Yaskawa INFORM job: vendrediTRJ3.JBI

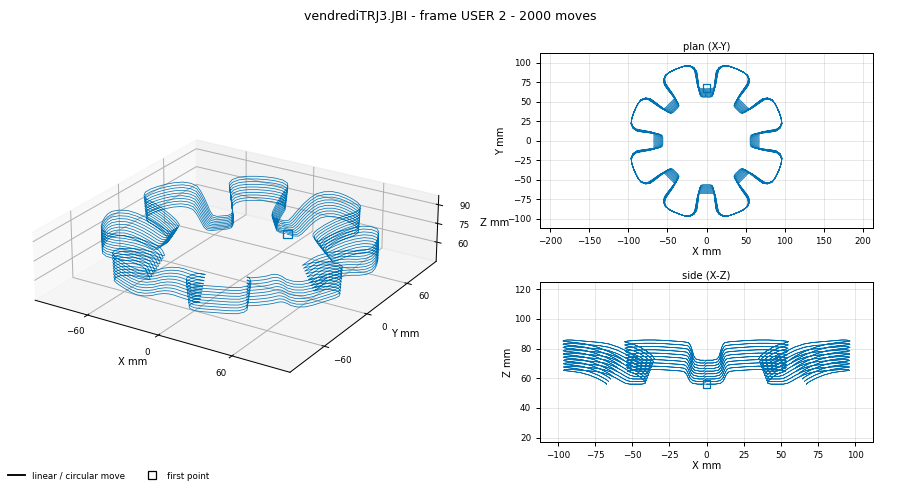
[picture p0: tool path of vendrediTRJ3.JBI in frame USER 2, 2000 of 2000 moves have a stored position in this frame; points joined in program order, loops and branches not executed]
/JOB
//NAME temp/vendrediTRJ3
///FOLDERNAME DEMO
//POS
///NPOS 2000,0,2000,0,0,0
///USER 2
///TOOL 7
///POSTYPE USER
///RECTAN
///RCONF 1,0,0,0,0,0,0,0,0,0,0,0,0,0,0,0,0,0,0,0,0,0,0,0
C00000=0.000,67.469,56.061,180.0000,38.4594,-10890.0000
C00001=2.820,67.413,56.044,-179.6998,38.4717,-10892.3954
C00002=5.989,67.263,56.069,174.6494,37.7561,-10895.0881
C00003=9.441,67.734,56.637,160.4399,22.8847,-10897.9350
C00004=11.191,69.937,58.076,177.3917,0.4478,-10899.0911
C00005=12.227,73.809,60.085,-176.5319,-0.2393,-10899.4060
C00006=13.183,79.025,62.181,-173.7887,-0.2511,-10899.4709
C00007=14.211,84.918,63.804,-172.0889,-0.3684,-10899.5004
C00008=15.500,90.396,64.610,-172.2474,-1.9783,-10899.7298
C00009=18.832,94.373,65.037,-176.4691,-3.4890,-10901.2851
C00010=23.832,96.213,65.385,-179.1427,-2.3150,-10903.9122
C00011=29.513,95.497,65.736,-179.9981,-0.1613,-10907.1736
C00012=35.347,93.539,65.969,-179.9993,-0.0181,-10910.7008
C00013=41.148,91.136,65.969,-179.9981,-0.0180,-10914.2992
C00014=46.658,88.395,65.736,179.9983,-0.1564,-10917.8267
C00015=51.181,84.885,65.385,179.1465,-2.3148,-10921.0877
C00016=53.416,80.048,65.037,176.4667,-3.4903,-10923.7152
C00017=52.959,74.880,64.610,172.2446,-1.9818,-10925.2699
C00018=49.997,70.095,63.804,172.0881,-0.3719,-10925.4993
C00019=46.557,65.200,62.181,173.7887,-0.2530,-10925.5293
C00020=43.545,60.837,60.085,176.5334,-0.2396,-10925.5938
C00021=41.540,57.367,58.076,-177.3875,0.4483,-10925.9087
C00022=41.220,54.571,56.637,-160.4399,22.8842,-10927.0654
C00023=43.327,51.796,56.069,-174.6518,37.7544,-10929.9123
C00024=45.674,49.662,56.044,179.7031,38.4687,-10932.6047
C00025=47.708,47.708,56.061,-180.0000,38.4581,-10935.0000
C00026=49.662,45.674,56.044,-179.7031,38.4687,-10937.3953
C00027=51.797,43.327,56.069,174.6514,37.7543,-10940.0883
C00028=54.571,41.220,56.637,160.4399,22.8842,-10942.9346
C00029=57.367,41.540,58.076,177.3875,0.4483,-10944.0913
C00030=60.837,43.545,60.085,-176.5334,-0.2396,-10944.4062
C00031=65.200,46.557,62.181,-173.7887,-0.2530,-10944.4707
C00032=70.095,49.997,63.804,-172.0881,-0.3719,-10944.5007
C00033=74.880,52.959,64.610,-172.2446,-1.9818,-10944.7301
C00034=80.048,53.416,65.037,-176.4667,-3.4903,-10946.2848
C00035=84.885,51.181,65.385,-179.1465,-2.3148,-10948.9123
C00036=88.395,46.658,65.736,-179.9983,-0.1564,-10952.1733
C00037=91.136,41.148,65.969,179.9981,-0.0180,-10955.7008
C00038=93.539,35.347,65.969,179.9993,-0.0181,-10959.2992
C00039=95.497,29.513,65.736,179.9981,-0.1613,-10962.8264
C00040=96.213,23.832,65.385,179.1427,-2.3150,-10966.0878
C00041=94.373,18.832,65.037,176.4691,-3.4890,-10968.7149
C00042=90.396,15.500,64.610,172.2474,-1.9783,-10970.2702
C00043=84.918,14.211,63.804,172.0889,-0.3684,-10970.4996
C00044=79.025,13.183,62.181,173.7887,-0.2511,-10970.5291
C00045=73.809,12.227,60.085,176.5319,-0.2393,-10970.5940
C00046=69.937,11.191,58.076,-177.3917,0.4478,-10970.9089
C00047=67.734,9.441,56.637,-160.4399,22.8847,-10972.0650
C00048=67.263,5.989,56.069,-174.6494,37.7561,-10974.9119
C00049=67.413,2.820,56.044,179.6998,38.4717,-10977.6046
C00050=67.469,0.000,56.061,-180.0000,38.4594,-10980.0000
C00051=67.413,-2.820,56.044,-179.6998,38.4717,-10982.3954
C00052=67.263,-5.989,56.069,174.6494,37.7561,-10985.0881
C00053=67.734,-9.441,56.637,160.4399,22.8847,-10987.9350
C00054=69.937,-11.191,58.076,177.3917,0.4478,-10989.0911
C00055=73.809,-12.227,60.085,-176.5319,-0.2393,-10989.4060
C00056=79.025,-13.183,62.181,-173.7887,-0.2511,-10989.4709
C00057=84.918,-14.211,63.804,-172.0889,-0.3684,-10989.5004
C00058=90.396,-15.500,64.610,-172.2474,-1.9783,-10989.7298
C00059=94.373,-18.832,65.037,-176.4691,-3.4890,-10991.2851
C00060=96.213,-23.832,65.385,-179.1427,-2.3150,-10993.9122
C00061=95.497,-29.513,65.736,-179.9981,-0.1613,-10997.1736
C00062=93.539,-35.347,65.969,-179.9993,-0.0181,-11000.7008
C00063=91.136,-41.148,65.969,-179.9981,-0.0180,-11004.2992
C00064=88.395,-46.658,65.736,179.9983,-0.1564,-11007.8267
C00065=84.885,-51.181,65.385,179.1465,-2.3148,-11011.0877
C00066=80.048,-53.416,65.037,176.4667,-3.4903,-11013.7152
C00067=74.880,-52.959,64.610,172.2446,-1.9818,-11015.2699
C00068=70.095,-49.997,63.804,172.0881,-0.3719,-11015.4993
C00069=65.200,-46.557,62.181,173.7887,-0.2530,-11015.5293
C00070=60.837,-43.545,60.085,176.5334,-0.2396,-11015.5938
C00071=57.367,-41.540,58.076,-177.3875,0.4483,-11015.9087
C00072=54.571,-41.220,56.637,-160.4399,22.8842,-11017.0654
C00073=51.796,-43.327,56.069,-174.6518,37.7544,-11019.9123
C00074=49.662,-45.674,56.044,179.7031,38.4687,-11022.6047
C00075=47.708,-47.708,56.061,-180.0000,38.4581,-11025.0000
C00076=45.674,-49.662,56.044,-179.7031,38.4687,-11027.3953
C00077=43.327,-51.797,56.069,174.6514,37.7543,-11030.0883
C00078=41.220,-54.571,56.637,160.4399,22.8842,-11032.9346
C00079=41.540,-57.367,58.076,177.3875,0.4483,-11034.0913
C00080=43.545,-60.837,60.085,-176.5334,-0.2396,-11034.4062
C00081=46.557,-65.200,62.181,-173.7887,-0.2530,-11034.4707
C00082=49.997,-70.095,63.804,-172.0881,-0.3719,-11034.5007
C00083=52.959,-74.880,64.610,-172.2446,-1.9818,-11034.7301
C00084=53.416,-80.048,65.037,-176.4667,-3.4903,-11036.2848
C00085=51.181,-84.885,65.385,-179.1465,-2.3148,-11038.9123
C00086=46.658,-88.395,65.736,-179.9983,-0.1564,-11042.1733
C00087=41.148,-91.136,65.969,179.9981,-0.0180,-11045.7008
C00088=35.347,-93.539,65.969,179.9993,-0.0181,-11049.2992
C00089=29.513,-95.497,65.736,179.9981,-0.1613,-11052.8264
C00090=23.832,-96.213,65.385,179.1427,-2.3150,-11056.0878
C00091=18.832,-94.373,65.037,176.4691,-3.4890,-11058.7149
C00092=15.500,-90.396,64.610,172.2474,-1.9783,-11060.2702
C00093=14.211,-84.918,63.804,172.0889,-0.3684,-11060.4996
C00094=13.183,-79.025,62.181,173.7887,-0.2511,-11060.5291
C00095=12.227,-73.809,60.085,176.5319,-0.2393,-11060.5940
C00096=11.191,-69.937,58.076,-177.3917,0.4478,-11060.9089
C00097=9.441,-67.734,56.637,-160.4399,22.8847,-11062.0650
C00098=5.989,-67.263,56.069,-174.6494,37.7561,-11064.9119
C00099=2.820,-67.413,56.044,179.6998,38.4717,-11067.6046
C00100=0.000,-67.469,56.061,-180.0000,38.4594,-11070.0000
C00101=-2.820,-67.413,56.044,-179.6998,38.4717,-11072.3954
C00102=-5.989,-67.263,56.069,174.6494,37.7561,-11075.0881
C00103=-9.441,-67.734,56.637,160.4399,22.8847,-11077.9350
C00104=-11.191,-69.937,58.076,177.3917,0.4478,-11079.0911
C00105=-12.227,-73.809,60.085,-176.5319,-0.2393,-11079.4060
C00106=-13.183,-79.025,62.181,-173.7887,-0.2511,-11079.4709
C00107=-14.211,-84.918,63.804,-172.0889,-0.3684,-11079.5004
C00108=-15.500,-90.396,64.610,-172.2474,-1.9783,-11079.7298
C00109=-18.832,-94.373,65.037,-176.4691,-3.4890,-11081.2851
C00110=-23.832,-96.213,65.385,-179.1427,-2.3150,-11083.9122
C00111=-29.513,-95.497,65.736,-179.9981,-0.1613,-11087.1736
C00112=-35.347,-93.539,65.969,-179.9993,-0.0181,-11090.7008
C00113=-41.148,-91.136,65.969,-179.9981,-0.0180,-11094.2992
C00114=-46.658,-88.395,65.736,179.9983,-0.1564,-11097.8267
C00115=-51.181,-84.885,65.385,179.1465,-2.3148,-11101.0877
C00116=-53.416,-80.048,65.037,176.4667,-3.4903,-11103.7152
C00117=-52.959,-74.880,64.610,172.2446,-1.9818,-11105.2699
C00118=-49.997,-70.095,63.804,172.0881,-0.3719,-11105.4993
C00119=-46.557,-65.200,62.181,173.7887,-0.2530,-11105.5293
C00120=-43.545,-60.837,60.085,176.5334,-0.2396,-11105.5938
C00121=-41.540,-57.367,58.076,-177.3875,0.4483,-11105.9087
C00122=-41.220,-54.571,56.637,-160.4399,22.8842,-11107.0654
C00123=-43.327,-51.796,56.069,-174.6518,37.7544,-11109.9123
C00124=-45.674,-49.662,56.044,179.7031,38.4687,-11112.6047
C00125=-47.708,-47.708,56.061,-180.0000,38.4581,-11115.0000
C00126=-49.662,-45.674,56.044,-179.7031,38.4687,-11117.3953
C00127=-51.797,-43.327,56.069,174.6514,37.7543,-11120.0883
C00128=-54.571,-41.220,56.637,160.4399,22.8842,-11122.9346
C00129=-57.367,-41.540,58.076,177.3875,0.4483,-11124.0913
C00130=-60.837,-43.545,60.085,-176.5334,-0.2396,-11124.4062
C00131=-65.200,-46.557,62.181,-173.7887,-0.2530,-11124.4707
C00132=-70.095,-49.997,63.804,-172.0881,-0.3719,-11124.5007
C00133=-74.880,-52.959,64.610,-172.2446,-1.9818,-11124.7301
C00134=-80.048,-53.416,65.037,-176.4667,-3.4903,-11126.2848
C00135=-84.885,-51.181,65.385,-179.1465,-2.3148,-11128.9123
C00136=-88.395,-46.658,65.736,-179.9983,-0.1564,-11132.1733
C00137=-91.136,-41.148,65.969,179.9981,-0.0180,-11135.7008
C00138=-93.539,-35.347,65.969,179.9993,-0.0181,-11139.2992
C00139=-95.497,-29.513,65.736,179.9981,-0.1613,-11142.8264
C00140=-96.213,-23.832,65.385,179.1427,-2.3150,-11146.0878
C00141=-94.373,-18.832,65.037,176.4691,-3.4890,-11148.7149
C00142=-90.396,-15.500,64.610,172.2474,-1.9783,-11150.2702
C00143=-84.918,-14.211,63.804,172.0889,-0.3684,-11150.4996
C00144=-79.025,-13.183,62.181,173.7887,-0.2511,-11150.5291
C00145=-73.809,-12.227,60.085,176.5319,-0.2393,-11150.5940
C00146=-69.937,-11.191,58.076,-177.3917,0.4478,-11150.9089
C00147=-67.734,-9.441,56.637,-160.4399,22.8847,-11152.0650
C00148=-67.263,-5.989,56.069,-174.6494,37.7561,-11154.9119
C00149=-67.413,-2.820,56.044,179.6998,38.4717,-11157.6046
C00150=-67.469,0.000,56.061,-180.0000,38.4594,-11160.0000
C00151=-67.413,2.820,56.044,-179.6998,38.4717,-11162.3954
C00152=-67.263,5.989,56.069,174.6494,37.7561,-11165.0881
C00153=-67.734,9.441,56.637,160.4399,22.8847,-11167.9350
C00154=-69.937,11.191,58.076,177.3917,0.4478,-11169.0911
C00155=-73.809,12.227,60.085,-176.5319,-0.2393,-11169.4060
C00156=-79.025,13.183,62.181,-173.7887,-0.2511,-11169.4709
C00157=-84.918,14.211,63.804,-172.0889,-0.3684,-11169.5004
C00158=-90.396,15.500,64.610,-172.2474,-1.9783,-11169.7298
C00159=-94.373,18.832,65.037,-176.4691,-3.4890,-11171.2851
C00160=-96.213,23.832,65.385,-179.1427,-2.3150,-11173.9122
C00161=-95.497,29.513,65.736,-179.9981,-0.1613,-11177.1736
C00162=-93.539,35.347,65.969,-179.9993,-0.0181,-11180.7008
C00163=-91.136,41.148,65.969,-179.9981,-0.0180,-11184.2992
C00164=-88.395,46.658,65.736,179.9983,-0.1564,-11187.8267
C00165=-84.885,51.181,65.385,179.1465,-2.3148,-11191.0877
C00166=-80.048,53.416,65.037,176.4667,-3.4903,-11193.7152
C00167=-74.880,52.959,64.610,172.2446,-1.9818,-11195.2699
C00168=-70.095,49.997,63.804,172.0881,-0.3719,-11195.4993
C00169=-65.200,46.557,62.181,173.7887,-0.2530,-11195.5293
C00170=-60.837,43.545,60.085,176.5334,-0.2396,-11195.5938
C00171=-57.367,41.540,58.076,-177.3875,0.4483,-11195.9087
C00172=-54.571,41.220,56.637,-160.4399,22.8842,-11197.0654
C00173=-51.796,43.327,56.069,-174.6518,37.7544,-11199.9123
C00174=-49.662,45.674,56.044,179.7031,38.4687,-11202.6047
C00175=-47.708,47.708,56.061,-180.0000,38.4581,-11205.0000
C00176=-45.674,49.662,56.044,-179.7031,38.4687,-11207.3953
C00177=-43.327,51.797,56.069,174.6514,37.7543,-11210.0883
C00178=-41.220,54.571,56.637,160.4399,22.8842,-11212.9346
C00179=-41.540,57.367,58.076,177.3875,0.4483,-11214.0913
C00180=-43.545,60.837,60.085,-176.5334,-0.2396,-11214.4062
C00181=-46.557,65.200,62.181,-173.7887,-0.2530,-11214.4707
C00182=-49.997,70.095,63.804,-172.0881,-0.3719,-11214.5007
C00183=-52.959,74.880,64.610,-172.2446,-1.9818,-11214.7301
C00184=-53.416,80.048,65.037,-176.4667,-3.4903,-11216.2848
C00185=-51.181,84.885,65.385,-179.1465,-2.3148,-11218.9123
C00186=-46.658,88.395,65.736,-179.9983,-0.1564,-11222.1733
C00187=-41.148,91.136,65.969,179.9981,-0.0180,-11225.7008
C00188=-35.347,93.539,65.969,179.9993,-0.0181,-11229.2992
C00189=-29.513,95.497,65.736,179.9981,-0.1613,-11232.8264
C00190=-23.832,96.213,65.385,179.1427,-2.3150,-11236.0878
C00191=-18.832,94.373,65.037,176.4691,-3.4890,-11238.7149
C00192=-15.500,90.396,64.610,172.2474,-1.9783,-11240.2702
C00193=-14.211,84.918,63.804,172.0889,-0.3684,-11240.4996
C00194=-13.183,79.025,62.181,173.7887,-0.2511,-11240.5291
C00195=-12.227,73.809,60.085,176.5319,-0.2393,-11240.5940
C00196=-11.191,69.937,58.076,-177.3917,0.4478,-11240.9089
C00197=-9.441,67.734,56.637,-160.4399,22.8847,-11242.0650
C00198=-5.989,67.263,56.069,-174.6494,37.7561,-11244.9119
C00199=-2.820,67.413,56.044,179.6998,38.4717,-11247.6046
C00200=0.000,66.107,57.788,180.0000,38.0594,-11250.0000
C00201=2.695,66.055,57.771,-179.6967,38.0667,-11252.3363
C00202=5.779,65.917,57.797,174.4231,37.2903,-11255.0104
C00203=9.185,66.436,58.394,160.6412,21.4973,-11257.8714
C00204=10.880,68.762,59.909,178.2705,0.2602,-11258.9912
C00205=11.874,72.826,62.021,-176.2283,-0.2219,-11259.2604
C00206=12.805,78.288,64.219,-173.7529,-0.2122,-11259.2892
C00207=13.814,84.445,65.915,-172.1933,-0.3031,-11259.2905
C00208=15.073,90.163,66.756,-172.3373,-1.8422,-11259.4907
C00209=18.432,94.325,67.200,-176.4590,-3.4166,-11261.0568
C00210=23.517,96.271,67.561,-179.1417,-2.2803,-11263.7273
C00211=29.315,95.562,67.927,179.9999,-0.1559,-11267.0541
C00212=35.280,93.564,68.167,-179.9993,-0.0181,-11270.6599
C00213=41.213,91.107,68.167,-179.9981,-0.0180,-11274.3400
C00214=46.844,88.301,67.927,179.9986,-0.1564,-11277.9461
C00215=51.445,84.703,67.561,179.1429,-2.2773,-11281.2727
C00216=53.664,79.731,67.200,176.4564,-3.4170,-11283.9430
C00217=53.097,74.413,66.756,172.3397,-1.8459,-11285.5096
C00218=49.944,69.479,65.915,172.1917,-0.3060,-11285.7099
C00219=46.303,64.413,64.219,173.7509,-0.2085,-11285.7103
C00220=43.100,59.892,62.021,176.2254,-0.2229,-11285.7399
C00221=40.929,56.315,59.909,-178.2687,0.2595,-11286.0092
C00222=40.483,53.472,58.394,-160.6426,21.4997,-11287.1289
C00223=42.524,50.697,57.797,-174.4236,37.2887,-11289.9895
C00224=44.802,48.614,57.771,179.6988,38.0662,-11292.6632
C00225=46.745,46.745,57.788,180.0000,38.0574,-11295.0000
C00226=48.613,44.802,57.771,-179.6984,38.0662,-11297.3362
C00227=50.697,42.524,57.797,174.4190,37.2852,-11300.0105
C00228=53.472,40.483,58.395,160.6426,21.4997,-11302.8711
C00229=56.315,40.929,59.909,178.2687,0.2595,-11303.9908
C00230=59.892,43.100,62.021,-176.2254,-0.2229,-11304.2601
C00231=64.413,46.303,64.219,-173.7509,-0.2085,-11304.2897
C00232=69.479,49.944,65.915,-172.1917,-0.3060,-11304.2901
C00233=74.413,53.097,66.756,-172.3397,-1.8459,-11304.4904
C00234=79.731,53.664,67.200,-176.4564,-3.4170,-11306.0570
C00235=84.703,51.445,67.561,-179.1429,-2.2773,-11308.7273
C00236=88.301,46.844,67.927,-179.9986,-0.1564,-11312.0539
C00237=91.107,41.213,68.167,179.9981,-0.0180,-11315.6600
C00238=93.564,35.280,68.167,179.9993,-0.0181,-11319.3401
C00239=95.562,29.315,67.927,-179.9999,-0.1559,-11322.9459
C00240=96.271,23.517,67.561,179.1417,-2.2803,-11326.2727
C00241=94.325,18.432,67.200,176.4590,-3.4166,-11328.9432
C00242=90.163,15.073,66.756,172.3373,-1.8422,-11330.5093
C00243=84.445,13.814,65.915,172.1933,-0.3031,-11330.7095
C00244=78.288,12.805,64.219,173.7529,-0.2122,-11330.7108
C00245=72.826,11.874,62.021,176.2283,-0.2219,-11330.7396
C00246=68.762,10.880,59.909,-178.2705,0.2602,-11331.0088
C00247=66.436,9.185,58.394,-160.6412,21.4973,-11332.1286
C00248=65.917,5.779,57.797,-174.4231,37.2903,-11334.9896
C00249=66.055,2.695,57.771,179.6967,38.0667,-11337.6637
C00250=66.107,0.000,57.788,180.0000,38.0594,-11340.0000
C00251=66.055,-2.695,57.771,-179.6967,38.0667,-11342.3363
C00252=65.917,-5.780,57.797,174.4154,37.2898,-11345.0112
C00253=66.436,-9.185,58.395,160.6412,21.4973,-11347.8714
C00254=68.762,-10.880,59.909,178.2705,0.2602,-11348.9912
C00255=72.826,-11.874,62.021,-176.2283,-0.2219,-11349.2604
C00256=78.288,-12.805,64.219,-173.7529,-0.2122,-11349.2892
C00257=84.445,-13.814,65.915,-172.1933,-0.3031,-11349.2905
C00258=90.163,-15.073,66.756,-172.3373,-1.8422,-11349.4907
C00259=94.325,-18.432,67.200,-176.4590,-3.4166,-11351.0568
C00260=96.271,-23.517,67.561,-179.1417,-2.2803,-11353.7273
C00261=95.562,-29.315,67.927,179.9999,-0.1559,-11357.0541
C00262=93.564,-35.280,68.167,-179.9993,-0.0181,-11360.6599
C00263=91.107,-41.213,68.167,-179.9981,-0.0180,-11364.3400
C00264=88.301,-46.844,67.927,179.9986,-0.1564,-11367.9461
C00265=84.703,-51.445,67.561,179.1429,-2.2773,-11371.2727
C00266=79.731,-53.664,67.200,176.4564,-3.4170,-11373.9430
C00267=74.413,-53.097,66.756,172.3397,-1.8459,-11375.5096
C00268=69.479,-49.944,65.915,172.1917,-0.3060,-11375.7099
C00269=64.413,-46.303,64.219,173.7509,-0.2085,-11375.7103
C00270=59.892,-43.100,62.021,176.2254,-0.2229,-11375.7399
C00271=56.315,-40.929,59.909,-178.2687,0.2595,-11376.0092
C00272=53.472,-40.483,58.394,-160.6426,21.4997,-11377.1289
C00273=50.697,-42.524,57.797,-174.4236,37.2887,-11379.9895
C00274=48.614,-44.802,57.771,179.6988,38.0662,-11382.6632
C00275=46.745,-46.745,57.788,180.0000,38.0574,-11385.0000
C00276=44.802,-48.613,57.771,-179.6984,38.0662,-11387.3362
C00277=42.524,-50.697,57.797,174.4190,37.2852,-11390.0105
C00278=40.483,-53.472,58.395,160.6426,21.4997,-11392.8711
C00279=40.929,-56.315,59.909,178.2687,0.2595,-11393.9908
C00280=43.100,-59.892,62.021,-176.2254,-0.2229,-11394.2601
C00281=46.303,-64.413,64.219,-173.7509,-0.2085,-11394.2897
C00282=49.944,-69.479,65.915,-172.1917,-0.3060,-11394.2901
C00283=53.097,-74.413,66.756,-172.3397,-1.8459,-11394.4904
C00284=53.664,-79.731,67.200,-176.4564,-3.4170,-11396.0570
C00285=51.445,-84.703,67.561,-179.1429,-2.2773,-11398.7273
C00286=46.844,-88.301,67.927,-179.9986,-0.1564,-11402.0539
C00287=41.213,-91.107,68.167,179.9981,-0.0180,-11405.6600
C00288=35.280,-93.564,68.167,179.9993,-0.0181,-11409.3401
C00289=29.315,-95.562,67.927,-179.9999,-0.1559,-11412.9459
C00290=23.517,-96.271,67.561,179.1417,-2.2803,-11416.2727
C00291=18.432,-94.325,67.200,176.4590,-3.4166,-11418.9432
C00292=15.073,-90.163,66.756,172.3373,-1.8422,-11420.5093
C00293=13.814,-84.445,65.915,172.1933,-0.3031,-11420.7095
C00294=12.805,-78.288,64.219,173.7529,-0.2122,-11420.7108
C00295=11.874,-72.826,62.021,176.2283,-0.2219,-11420.7396
C00296=10.880,-68.762,59.909,-178.2705,0.2602,-11421.0088
C00297=9.185,-66.436,58.394,-160.6412,21.4973,-11422.1286
C00298=5.779,-65.917,57.797,-174.4231,37.2903,-11424.9896
C00299=2.695,-66.055,57.771,179.6967,38.0667,-11427.6637
C00300=0.000,-66.107,57.788,-180.0000,38.0594,-11430.0000
C00301=-2.695,-66.055,57.771,-179.6967,38.0667,-11432.3363
C00302=-5.780,-65.917,57.797,174.4154,37.2898,-11435.0112
C00303=-9.185,-66.436,58.395,160.6412,21.4973,-11437.8714
C00304=-10.880,-68.762,59.909,178.2705,0.2602,-11438.9912
C00305=-11.874,-72.826,62.021,-176.2283,-0.2219,-11439.2604
C00306=-12.805,-78.288,64.219,-173.7529,-0.2122,-11439.2892
C00307=-13.814,-84.445,65.915,-172.1933,-0.3031,-11439.2905
C00308=-15.073,-90.163,66.756,-172.3373,-1.8422,-11439.4907
C00309=-18.432,-94.325,67.200,-176.4590,-3.4166,-11441.0568
C00310=-23.517,-96.271,67.561,-179.1417,-2.2803,-11443.7273
C00311=-29.315,-95.562,67.927,179.9999,-0.1559,-11447.0541
C00312=-35.280,-93.564,68.167,-179.9993,-0.0181,-11450.6599
C00313=-41.213,-91.107,68.167,-179.9981,-0.0180,-11454.3400
C00314=-46.844,-88.301,67.927,179.9986,-0.1564,-11457.9461
C00315=-51.445,-84.703,67.561,179.1429,-2.2773,-11461.2727
C00316=-53.664,-79.731,67.200,176.4564,-3.4170,-11463.9430
C00317=-53.097,-74.413,66.756,172.3397,-1.8459,-11465.5096
C00318=-49.944,-69.479,65.915,172.1917,-0.3060,-11465.7099
C00319=-46.303,-64.413,64.219,173.7509,-0.2085,-11465.7103
C00320=-43.100,-59.892,62.021,176.2254,-0.2229,-11465.7399
C00321=-40.929,-56.315,59.909,-178.2687,0.2595,-11466.0092
C00322=-40.483,-53.472,58.394,-160.6426,21.4997,-11467.1289
C00323=-42.524,-50.697,57.797,-174.4236,37.2887,-11469.9895
C00324=-44.802,-48.614,57.771,179.6988,38.0662,-11472.6632
C00325=-46.745,-46.745,57.788,-180.0000,38.0574,-11475.0000
C00326=-48.613,-44.802,57.771,-179.6984,38.0662,-11477.3362
C00327=-50.697,-42.524,57.797,174.4190,37.2852,-11480.0105
C00328=-53.472,-40.483,58.395,160.6426,21.4997,-11482.8711
C00329=-56.315,-40.929,59.909,178.2687,0.2595,-11483.9908
C00330=-59.892,-43.100,62.021,-176.2254,-0.2229,-11484.2601
C00331=-64.413,-46.303,64.219,-173.7509,-0.2085,-11484.2897
C00332=-69.479,-49.944,65.915,-172.1917,-0.3060,-11484.2901
C00333=-74.413,-53.097,66.756,-172.3397,-1.8459,-11484.4904
C00334=-79.731,-53.664,67.200,-176.4564,-3.4170,-11486.0570
C00335=-84.703,-51.445,67.561,-179.1429,-2.2773,-11488.7273
C00336=-88.301,-46.844,67.927,-179.9986,-0.1564,-11492.0539
C00337=-91.107,-41.213,68.167,179.9981,-0.0180,-11495.6600
C00338=-93.564,-35.280,68.167,179.9993,-0.0181,-11499.3401
C00339=-95.562,-29.315,67.927,-179.9999,-0.1559,-11502.9459
C00340=-96.271,-23.517,67.561,179.1417,-2.2803,-11506.2727
C00341=-94.325,-18.432,67.200,176.4590,-3.4166,-11508.9432
C00342=-90.163,-15.073,66.756,172.3373,-1.8422,-11510.5093
C00343=-84.445,-13.814,65.915,172.1933,-0.3031,-11510.7095
C00344=-78.288,-12.805,64.219,173.7529,-0.2122,-11510.7108
C00345=-72.826,-11.874,62.021,176.2283,-0.2219,-11510.7396
C00346=-68.762,-10.880,59.909,-178.2705,0.2602,-11511.0088
C00347=-66.436,-9.185,58.394,-160.6412,21.4973,-11512.1286
C00348=-65.917,-5.779,57.797,-174.4231,37.2903,-11514.9896
C00349=-66.055,-2.695,57.771,179.6967,38.0667,-11517.6637
C00350=-66.107,0.000,57.788,-180.0000,38.0594,-11520.0000
C00351=-66.055,2.695,57.771,-179.6967,38.0667,-11522.3363
C00352=-65.917,5.780,57.797,174.4154,37.2898,-11525.0112
C00353=-66.436,9.185,58.395,160.6412,21.4973,-11527.8714
C00354=-68.762,10.880,59.909,178.2705,0.2602,-11528.9912
C00355=-72.826,11.874,62.021,-176.2283,-0.2219,-11529.2604
C00356=-78.288,12.805,64.219,-173.7529,-0.2122,-11529.2892
C00357=-84.445,13.814,65.915,-172.1933,-0.3031,-11529.2905
C00358=-90.163,15.073,66.756,-172.3373,-1.8422,-11529.4907
C00359=-94.325,18.432,67.200,-176.4590,-3.4166,-11531.0568
C00360=-96.271,23.517,67.561,-179.1417,-2.2803,-11533.7273
C00361=-95.562,29.315,67.927,179.9999,-0.1559,-11537.0541
C00362=-93.564,35.280,68.167,-179.9993,-0.0181,-11540.6599
C00363=-91.107,41.213,68.167,-179.9981,-0.0180,-11544.3400
C00364=-88.301,46.844,67.927,179.9986,-0.1564,-11547.9461
C00365=-84.703,51.445,67.561,179.1429,-2.2773,-11551.2727
C00366=-79.731,53.664,67.200,176.4564,-3.4170,-11553.9430
C00367=-74.413,53.097,66.756,172.3397,-1.8459,-11555.5096
C00368=-69.479,49.944,65.915,172.1917,-0.3060,-11555.7099
C00369=-64.413,46.303,64.219,173.7509,-0.2085,-11555.7103
C00370=-59.892,43.100,62.021,176.2254,-0.2229,-11555.7399
C00371=-56.315,40.929,59.909,-178.2687,0.2595,-11556.0092
C00372=-53.472,40.483,58.394,-160.6426,21.4997,-11557.1289
C00373=-50.697,42.524,57.797,-174.4236,37.2887,-11559.9895
C00374=-48.614,44.802,57.771,179.6988,38.0662,-11562.6632
C00375=-46.745,46.745,57.788,-180.0000,38.0574,-11565.0000
C00376=-44.802,48.613,57.771,-179.6984,38.0662,-11567.3362
C00377=-42.524,50.697,57.797,174.4190,37.2852,-11570.0105
C00378=-40.483,53.472,58.395,160.6426,21.4997,-11572.8711
C00379=-40.929,56.315,59.909,178.2687,0.2595,-11573.9908
C00380=-43.100,59.892,62.021,-176.2254,-0.2229,-11574.2601
C00381=-46.303,64.413,64.219,-173.7509,-0.2085,-11574.2897
C00382=-49.944,69.479,65.915,-172.1917,-0.3060,-11574.2901
C00383=-53.097,74.413,66.756,-172.3397,-1.8459,-11574.4904
C00384=-53.664,79.731,67.200,-176.4564,-3.4170,-11576.0570
C00385=-51.445,84.703,67.561,-179.1429,-2.2773,-11578.7273
C00386=-46.844,88.301,67.927,-179.9986,-0.1564,-11582.0539
C00387=-41.213,91.107,68.167,179.9981,-0.0180,-11585.6600
C00388=-35.280,93.564,68.167,179.9993,-0.0181,-11589.3401
C00389=-29.315,95.562,67.927,-179.9999,-0.1559,-11592.9459
C00390=-23.517,96.271,67.561,179.1417,-2.2803,-11596.2727
C00391=-18.432,94.325,67.200,176.4590,-3.4166,-11598.9432
C00392=-15.073,90.163,66.756,172.3373,-1.8422,-11600.5093
C00393=-13.814,84.445,65.915,172.1933,-0.3031,-11600.7095
C00394=-12.805,78.288,64.219,173.7529,-0.2122,-11600.7108
C00395=-11.874,72.826,62.021,176.2283,-0.2219,-11600.7396
C00396=-10.880,68.762,59.909,-178.2705,0.2602,-11601.0088
C00397=-9.185,66.436,58.395,-160.6412,21.4973,-11602.1286
C00398=-5.780,65.917,57.797,-174.4154,37.2898,-11604.9888
C00399=-2.695,66.055,57.771,179.6967,38.0667,-11607.6637
C00400=0.000,64.758,59.526,-180.0000,37.5735,-11610.0000
C00401=2.572,64.710,59.508,-179.6979,37.5837,-11612.2761
C00402=5.572,64.584,59.535,174.2146,36.7296,-11614.9310
C00403=8.932,65.152,60.163,160.9703,20.0908,-11617.8063
C00404=10.572,67.603,61.754,179.0583,0.1253,-11618.8881
C00405=11.527,71.864,63.969,-175.9897,-0.1992,-11619.1126
C00406=12.439,77.571,66.266,-173.7747,-0.1711,-11619.1102
C00407=13.430,83.988,68.033,-172.3612,-0.2407,-11619.0849
C00408=14.662,89.940,68.906,-172.5060,-1.7115,-11619.2589
C00409=18.048,94.279,69.366,-176.4898,-3.3102,-11620.8371
C00410=23.215,96.325,69.740,-179.1510,-2.2246,-11623.5503
C00411=29.126,95.625,70.117,179.9996,-0.1559,-11626.9400
C00412=35.216,93.589,70.366,-179.9993,-0.0181,-11630.6205
C00413=41.276,91.079,70.366,-179.9981,-0.0180,-11634.3795
C00414=47.022,88.212,70.117,179.9990,-0.1564,-11638.0601
C00415=51.697,84.528,69.740,179.1554,-2.2229,-11641.4498
C00416=53.903,79.427,69.366,176.4883,-3.3136,-11644.1627
C00417=53.229,73.964,68.906,172.5034,-1.7072,-11645.7411
C00418=49.892,68.885,68.033,172.3610,-0.2408,-11645.9150
C00419=46.056,63.647,66.266,173.7731,-0.1698,-11645.8901
C00420=42.664,58.966,63.969,175.9921,-0.2034,-11645.8871
C00421=40.327,55.279,61.754,-179.0540,0.1227,-11646.1114
C00422=39.754,52.385,60.163,-160.9694,20.0893,-11647.1942
C00423=41.728,49.608,59.535,-174.2183,36.7311,-11650.0690
C00424=43.938,47.576,59.508,179.6961,37.5811,-11652.7235
C00425=45.791,45.791,59.526,-180.0000,37.5739,-11655.0000
C00426=47.575,43.938,59.508,-179.6957,37.5811,-11657.2759
C00427=49.608,41.728,59.535,174.2083,36.7306,-11659.9310
C00428=52.385,39.754,60.163,160.9694,20.0893,-11662.8058
C00429=55.279,40.327,61.754,179.0540,0.1227,-11663.8886
C00430=58.966,42.664,63.969,-175.9921,-0.2034,-11664.1129
C00431=63.647,46.056,66.266,-173.7731,-0.1698,-11664.1099
C00432=68.885,49.892,68.033,-172.3610,-0.2408,-11664.0850
C00433=73.964,53.229,68.906,-172.5034,-1.7072,-11664.2589
C00434=79.427,53.903,69.366,-176.4883,-3.3136,-11665.8373
C00435=84.528,51.697,69.740,-179.1554,-2.2229,-11668.5502
C00436=88.212,47.022,70.117,-179.9990,-0.1564,-11671.9399
C00437=91.079,41.276,70.366,179.9981,-0.0180,-11675.6205
C00438=93.589,35.216,70.366,179.9993,-0.0181,-11679.3795
C00439=95.625,29.126,70.117,-179.9996,-0.1559,-11683.0600
C00440=96.325,23.215,69.740,179.1510,-2.2246,-11686.4497
C00441=94.279,18.048,69.366,176.4898,-3.3102,-11689.1629
C00442=89.940,14.662,68.906,172.5060,-1.7115,-11690.7411
C00443=83.988,13.430,68.033,172.3612,-0.2407,-11690.9151
C00444=77.571,12.439,66.266,173.7747,-0.1711,-11690.8898
C00445=71.864,11.527,63.969,175.9897,-0.1992,-11690.8874
C00446=67.603,10.572,61.754,-179.0583,0.1253,-11691.1119
C00447=65.152,8.932,60.163,-160.9703,20.0908,-11692.1937
C00448=64.584,5.572,59.535,-174.2146,36.7296,-11695.0690
C00449=64.710,2.572,59.508,179.6979,37.5837,-11697.7239
C00450=64.758,0.000,59.526,180.0000,37.5735,-11700.0000
C00451=64.710,-2.572,59.508,-179.6979,37.5837,-11702.2761
C00452=64.584,-5.572,59.535,174.2146,36.7296,-11704.9310
C00453=65.152,-8.932,60.163,160.9703,20.0908,-11707.8063
C00454=67.603,-10.572,61.754,179.0583,0.1253,-11708.8881
C00455=71.864,-11.527,63.969,-175.9897,-0.1992,-11709.1126
C00456=77.571,-12.439,66.266,-173.7747,-0.1711,-11709.1102
C00457=83.988,-13.430,68.033,-172.3612,-0.2407,-11709.0849
C00458=89.940,-14.662,68.906,-172.5060,-1.7115,-11709.2589
C00459=94.279,-18.048,69.366,-176.4898,-3.3102,-11710.8371
C00460=96.325,-23.215,69.740,-179.1510,-2.2246,-11713.5503
C00461=95.625,-29.126,70.117,179.9996,-0.1559,-11716.9400
C00462=93.589,-35.216,70.366,-179.9993,-0.0181,-11720.6205
C00463=91.079,-41.276,70.366,-179.9981,-0.0180,-11724.3795
C00464=88.212,-47.022,70.117,179.9990,-0.1564,-11728.0601
C00465=84.528,-51.697,69.740,179.1554,-2.2229,-11731.4498
C00466=79.427,-53.903,69.366,176.4883,-3.3136,-11734.1627
C00467=73.964,-53.229,68.906,172.5034,-1.7072,-11735.7411
C00468=68.885,-49.892,68.033,172.3610,-0.2408,-11735.9150
C00469=63.647,-46.056,66.266,173.7731,-0.1698,-11735.8901
C00470=58.966,-42.664,63.969,175.9921,-0.2034,-11735.8871
C00471=55.279,-40.327,61.754,-179.0540,0.1227,-11736.1114
C00472=52.385,-39.754,60.163,-160.9694,20.0893,-11737.1942
C00473=49.608,-41.728,59.535,-174.2183,36.7311,-11740.0690
C00474=47.576,-43.938,59.508,179.6961,37.5811,-11742.7235
C00475=45.791,-45.791,59.526,180.0000,37.5739,-11745.0000
C00476=43.938,-47.575,59.508,-179.6957,37.5811,-11747.2759
C00477=41.728,-49.608,59.535,174.2083,36.7306,-11749.9310
C00478=39.754,-52.385,60.163,160.9694,20.0893,-11752.8058
C00479=40.327,-55.279,61.754,179.0540,0.1227,-11753.8886
C00480=42.664,-58.966,63.969,-175.9921,-0.2034,-11754.1129
C00481=46.056,-63.647,66.266,-173.7731,-0.1698,-11754.1099
C00482=49.892,-68.885,68.033,-172.3610,-0.2408,-11754.0850
C00483=53.229,-73.964,68.906,-172.5034,-1.7072,-11754.2589
C00484=53.903,-79.427,69.366,-176.4883,-3.3136,-11755.8373
C00485=51.697,-84.528,69.740,-179.1554,-2.2229,-11758.5502
C00486=47.022,-88.212,70.117,-179.9990,-0.1564,-11761.9399
C00487=41.276,-91.079,70.366,179.9981,-0.0180,-11765.6205
C00488=35.216,-93.589,70.366,179.9993,-0.0181,-11769.3795
C00489=29.126,-95.625,70.117,-179.9996,-0.1559,-11773.0600
C00490=23.215,-96.325,69.740,179.1510,-2.2246,-11776.4497
C00491=18.048,-94.279,69.366,176.4898,-3.3102,-11779.1629
C00492=14.662,-89.940,68.906,172.5060,-1.7115,-11780.7411
C00493=13.430,-83.988,68.033,172.3612,-0.2407,-11780.9151
C00494=12.439,-77.571,66.266,173.7747,-0.1711,-11780.8898
C00495=11.527,-71.864,63.969,175.9897,-0.1992,-11780.8874
C00496=10.572,-67.603,61.754,-179.0583,0.1253,-11781.1119
C00497=8.932,-65.152,60.163,-160.9703,20.0908,-11782.1937
C00498=5.572,-64.584,59.535,-174.2146,36.7296,-11785.0690
C00499=2.572,-64.710,59.508,179.6979,37.5837,-11787.7239
C00500=0.000,-64.758,59.526,180.0000,37.5735,-11790.0000
C00501=-2.572,-64.710,59.508,-179.6979,37.5837,-11792.2761
C00502=-5.572,-64.584,59.535,174.2146,36.7296,-11794.9310
C00503=-8.932,-65.152,60.163,160.9703,20.0908,-11797.8063
C00504=-10.572,-67.603,61.754,179.0583,0.1253,-11798.8881
C00505=-11.527,-71.864,63.969,-175.9897,-0.1992,-11799.1126
C00506=-12.439,-77.571,66.266,-173.7747,-0.1711,-11799.1102
C00507=-13.430,-83.988,68.033,-172.3612,-0.2407,-11799.0849
C00508=-14.662,-89.940,68.906,-172.5060,-1.7115,-11799.2589
C00509=-18.048,-94.279,69.366,-176.4898,-3.3102,-11800.8371
C00510=-23.215,-96.325,69.740,-179.1510,-2.2246,-11803.5503
C00511=-29.126,-95.625,70.117,179.9996,-0.1559,-11806.9400
C00512=-35.216,-93.589,70.366,-179.9993,-0.0181,-11810.6205
C00513=-41.276,-91.079,70.366,-179.9981,-0.0180,-11814.3795
C00514=-47.022,-88.212,70.117,179.9990,-0.1564,-11818.0601
C00515=-51.697,-84.528,69.740,179.1554,-2.2229,-11821.4498
C00516=-53.903,-79.427,69.366,176.4883,-3.3136,-11824.1627
C00517=-53.229,-73.964,68.906,172.5034,-1.7072,-11825.7411
C00518=-49.892,-68.885,68.033,172.3610,-0.2408,-11825.9150
C00519=-46.056,-63.647,66.266,173.7731,-0.1698,-11825.8901
C00520=-42.664,-58.966,63.969,175.9921,-0.2034,-11825.8871
C00521=-40.327,-55.279,61.754,-179.0540,0.1227,-11826.1114
C00522=-39.754,-52.385,60.163,-160.9694,20.0893,-11827.1942
C00523=-41.728,-49.608,59.535,-174.2183,36.7311,-11830.0690
C00524=-43.938,-47.576,59.508,179.6961,37.5811,-11832.7235
C00525=-45.791,-45.791,59.526,180.0000,37.5739,-11835.0000
C00526=-47.575,-43.938,59.508,-179.6957,37.5811,-11837.2759
C00527=-49.608,-41.728,59.535,174.2083,36.7306,-11839.9310
C00528=-52.385,-39.754,60.163,160.9694,20.0893,-11842.8058
C00529=-55.279,-40.327,61.754,179.0540,0.1227,-11843.8886
C00530=-58.966,-42.664,63.969,-175.9921,-0.2034,-11844.1129
C00531=-63.647,-46.056,66.266,-173.7731,-0.1698,-11844.1099
C00532=-68.885,-49.892,68.033,-172.3610,-0.2408,-11844.0850
C00533=-73.964,-53.229,68.906,-172.5034,-1.7072,-11844.2589
C00534=-79.427,-53.903,69.366,-176.4883,-3.3136,-11845.8373
C00535=-84.528,-51.697,69.740,-179.1554,-2.2229,-11848.5502
C00536=-88.212,-47.022,70.117,-179.9990,-0.1564,-11851.9399
C00537=-91.079,-41.276,70.366,179.9981,-0.0180,-11855.6205
C00538=-93.589,-35.216,70.366,179.9993,-0.0181,-11859.3795
C00539=-95.625,-29.126,70.117,-179.9996,-0.1559,-11863.0600
C00540=-96.325,-23.215,69.740,179.1510,-2.2246,-11866.4497
C00541=-94.279,-18.048,69.366,176.4898,-3.3102,-11869.1629
C00542=-89.940,-14.662,68.906,172.5060,-1.7115,-11870.7411
C00543=-83.988,-13.430,68.033,172.3612,-0.2407,-11870.9151
C00544=-77.571,-12.439,66.266,173.7747,-0.1711,-11870.8898
C00545=-71.864,-11.527,63.969,175.9897,-0.1992,-11870.8874
C00546=-67.603,-10.572,61.754,-179.0583,0.1253,-11871.1119
C00547=-65.152,-8.932,60.163,-160.9703,20.0908,-11872.1937
C00548=-64.584,-5.572,59.535,-174.2146,36.7296,-11875.0690
C00549=-64.710,-2.572,59.508,179.6979,37.5837,-11877.7239
C00550=-64.758,0.000,59.526,-180.0000,37.5735,-11880.0000
C00551=-64.710,2.572,59.508,-179.6979,37.5837,-11882.2761
C00552=-64.584,5.572,59.535,174.2146,36.7296,-11884.9310
C00553=-65.152,8.932,60.163,160.9703,20.0908,-11887.8063
C00554=-67.603,10.572,61.754,179.0583,0.1253,-11888.8881
C00555=-71.864,11.527,63.969,-175.9897,-0.1992,-11889.1126
C00556=-77.571,12.439,66.266,-173.7747,-0.1711,-11889.1102
C00557=-83.988,13.430,68.033,-172.3612,-0.2407,-11889.0849
C00558=-89.940,14.662,68.906,-172.5060,-1.7115,-11889.2589
C00559=-94.279,18.048,69.366,-176.4898,-3.3102,-11890.8371
C00560=-96.325,23.215,69.740,-179.1510,-2.2246,-11893.5503
C00561=-95.625,29.126,70.117,179.9996,-0.1559,-11896.9400
C00562=-93.589,35.216,70.366,-179.9993,-0.0181,-11900.6205
C00563=-91.079,41.276,70.366,-179.9981,-0.0180,-11904.3795
C00564=-88.212,47.022,70.117,179.9990,-0.1564,-11908.0601
C00565=-84.528,51.697,69.740,179.1554,-2.2229,-11911.4498
C00566=-79.427,53.903,69.366,176.4883,-3.3136,-11914.1627
C00567=-73.964,53.229,68.906,172.5034,-1.7072,-11915.7411
C00568=-68.885,49.892,68.033,172.3610,-0.2408,-11915.9150
C00569=-63.647,46.056,66.266,173.7731,-0.1698,-11915.8901
C00570=-58.966,42.664,63.969,175.9921,-0.2034,-11915.8871
C00571=-55.279,40.327,61.754,-179.0540,0.1227,-11916.1114
C00572=-52.385,39.754,60.163,-160.9694,20.0893,-11917.1942
C00573=-49.608,41.728,59.535,-174.2183,36.7311,-11920.0690
C00574=-47.576,43.938,59.508,179.6961,37.5811,-11922.7235
C00575=-45.791,45.791,59.526,-180.0000,37.5739,-11925.0000
C00576=-43.938,47.575,59.508,-179.6957,37.5811,-11927.2759
C00577=-41.728,49.608,59.535,174.2083,36.7306,-11929.9310
C00578=-39.754,52.385,60.163,160.9694,20.0893,-11932.8058
C00579=-40.327,55.279,61.754,179.0540,0.1227,-11933.8886
C00580=-42.664,58.966,63.969,-175.9921,-0.2034,-11934.1129
C00581=-46.056,63.647,66.266,-173.7731,-0.1698,-11934.1099
C00582=-49.892,68.885,68.033,-172.3610,-0.2408,-11934.0850
C00583=-53.229,73.964,68.906,-172.5034,-1.7072,-11934.2589
C00584=-53.903,79.427,69.366,-176.4883,-3.3136,-11935.8373
C00585=-51.697,84.528,69.740,-179.1554,-2.2229,-11938.5502
C00586=-47.022,88.212,70.117,-179.9990,-0.1564,-11941.9399
C00587=-41.276,91.079,70.366,179.9981,-0.0180,-11945.6205
C00588=-35.216,93.589,70.366,179.9993,-0.0181,-11949.3795
C00589=-29.126,95.625,70.117,-179.9996,-0.1559,-11953.0600
C00590=-23.215,96.325,69.740,179.1510,-2.2246,-11956.4497
C00591=-18.048,94.279,69.366,176.4898,-3.3102,-11959.1629
C00592=-14.662,89.940,68.906,172.5060,-1.7115,-11960.7411
C00593=-13.430,83.988,68.033,172.3612,-0.2407,-11960.9151
C00594=-12.439,77.571,66.266,173.7747,-0.1711,-11960.8898
C00595=-11.527,71.864,63.969,175.9897,-0.1992,-11960.8874
C00596=-10.572,67.603,61.754,-179.0583,0.1253,-11961.1119
C00597=-8.932,65.152,60.163,-160.9703,20.0908,-11962.1937
C00598=-5.572,64.584,59.535,-174.2146,36.7296,-11965.0690
C00599=-2.572,64.710,59.508,179.6979,37.5837,-11967.7239
C00600=0.000,63.425,61.276,-180.0000,37.0005,-11970.0000
C00601=2.450,63.381,61.257,-179.6948,37.0092,-11972.2137
C00602=5.367,63.268,61.285,174.0310,36.0790,-11974.8488
C00603=8.682,63.886,61.945,161.4111,18.6823,-11977.7390
C00604=10.270,66.465,63.612,179.7526,0.0255,-11978.7837
C00605=11.189,70.924,65.929,-175.8210,-0.1771,-11978.9651
C00606=12.084,76.878,68.324,-173.8594,-0.1394,-11978.9329
C00607=13.063,83.550,70.157,-172.5965,-0.1926,-11978.8862
C00608=14.270,89.726,71.060,-172.7438,-1.5775,-11979.0366
C00609=17.683,94.235,71.535,-176.5649,-3.1765,-11980.6278
C00610=22.929,96.378,71.920,-179.1719,-2.1420,-11983.3823
C00611=28.946,95.684,72.309,-179.9969,-0.1487,-11986.8314
C00612=35.156,93.612,72.565,-179.9993,-0.0181,-11990.5837
C00613=41.335,91.053,72.565,-179.9981,-0.0180,-11994.4165
C00614=47.191,88.127,72.309,179.9965,-0.1513,-11998.1685
C00615=51.936,84.362,71.920,179.1729,-2.1445,-12001.6178
C00616=54.130,79.138,71.535,176.5613,-3.1804,-12004.3719
C00617=53.356,73.536,71.060,172.7432,-1.5739,-12005.9638
C00618=49.842,68.316,70.157,172.5980,-0.1884,-12006.1137
C00619=45.816,62.906,68.324,173.8645,-0.1373,-12006.0668
C00620=42.239,58.063,65.929,175.8220,-0.1746,-12006.0347
C00621=39.736,54.260,63.612,-179.7499,0.0269,-12006.2163
C00622=39.035,51.313,61.945,-161.4145,18.6787,-12007.2611
C00623=40.942,48.532,61.285,-174.0315,36.0780,-12010.1513
C00624=43.085,46.550,61.257,179.6995,37.0101,-12012.7862
C00625=44.848,44.848,61.276,-180.0000,36.9982,-12015.0000
C00626=46.550,43.085,61.257,-179.6995,37.0101,-12017.2138
C00627=48.532,40.942,61.285,174.0315,36.0780,-12019.8487
C00628=51.313,39.035,61.945,161.4145,18.6787,-12022.7389
C00629=54.260,39.736,63.612,179.7499,0.0269,-12023.7837
C00630=58.063,42.239,65.929,-175.8220,-0.1746,-12023.9653
C00631=62.906,45.816,68.324,-173.8645,-0.1373,-12023.9332
C00632=68.316,49.842,70.157,-172.5980,-0.1884,-12023.8863
C00633=73.536,53.356,71.060,-172.7432,-1.5739,-12024.0362
C00634=79.138,54.130,71.535,-176.5613,-3.1804,-12025.6281
C00635=84.362,51.936,71.920,-179.1729,-2.1445,-12028.3822
C00636=88.127,47.191,72.309,-179.9965,-0.1513,-12031.8315
C00637=91.053,41.335,72.565,179.9981,-0.0180,-12035.5835
C00638=93.612,35.156,72.565,179.9993,-0.0181,-12039.4163
C00639=95.684,28.946,72.309,179.9969,-0.1487,-12043.1686
C00640=96.378,22.929,71.920,179.1719,-2.1420,-12046.6177
C00641=94.235,17.683,71.535,176.5649,-3.1765,-12049.3722
C00642=89.726,14.270,71.060,172.7438,-1.5775,-12050.9634
C00643=83.550,13.063,70.157,172.5965,-0.1926,-12051.1138
C00644=76.878,12.084,68.324,173.8594,-0.1394,-12051.0671
C00645=70.924,11.189,65.929,175.8210,-0.1771,-12051.0349
C00646=66.465,10.270,63.612,-179.7526,0.0255,-12051.2163
C00647=63.886,8.682,61.945,-161.4111,18.6823,-12052.2610
C00648=63.268,5.367,61.285,-174.0310,36.0790,-12055.1512
C00649=63.381,2.450,61.257,179.6948,37.0092,-12057.7863
C00650=63.425,0.000,61.276,-180.0000,37.0005,-12060.0000
C00651=63.381,-2.450,61.257,-179.6948,37.0092,-12062.2137
C00652=63.268,-5.367,61.285,174.0310,36.0790,-12064.8488
C00653=63.886,-8.682,61.945,161.4119,18.6766,-12067.7390
C00654=66.465,-10.270,63.612,179.7526,0.0255,-12068.7837
C00655=70.924,-11.189,65.929,-175.8210,-0.1771,-12068.9651
C00656=76.878,-12.084,68.324,-173.8594,-0.1394,-12068.9329
C00657=83.550,-13.063,70.157,-172.5965,-0.1926,-12068.8862
C00658=89.726,-14.270,71.060,-172.7438,-1.5775,-12069.0366
C00659=94.235,-17.683,71.535,-176.5649,-3.1765,-12070.6278
C00660=96.378,-22.929,71.920,-179.1719,-2.1420,-12073.3823
C00661=95.684,-28.946,72.309,-179.9969,-0.1487,-12076.8314
C00662=93.612,-35.156,72.565,-179.9993,-0.0181,-12080.5837
C00663=91.053,-41.335,72.565,-179.9981,-0.0180,-12084.4165
C00664=88.127,-47.191,72.309,179.9965,-0.1513,-12088.1685
C00665=84.362,-51.936,71.920,179.1729,-2.1445,-12091.6178
C00666=79.138,-54.130,71.535,176.5613,-3.1804,-12094.3719
C00667=73.536,-53.356,71.060,172.7432,-1.5739,-12095.9638
C00668=68.316,-49.842,70.157,172.5980,-0.1884,-12096.1137
C00669=62.906,-45.816,68.324,173.8645,-0.1373,-12096.0668
C00670=58.063,-42.239,65.929,175.8220,-0.1746,-12096.0347
C00671=54.260,-39.736,63.612,-179.7499,0.0269,-12096.2163
C00672=51.313,-39.035,61.945,-161.4145,18.6787,-12097.2611
C00673=48.532,-40.942,61.285,-174.0315,36.0780,-12100.1513
C00674=46.550,-43.085,61.257,179.6995,37.0101,-12102.7862
C00675=44.848,-44.848,61.276,-180.0000,36.9982,-12105.0000
C00676=43.085,-46.550,61.257,-179.6995,37.0101,-12107.2138
C00677=40.942,-48.532,61.285,174.0315,36.0780,-12109.8487
C00678=39.035,-51.313,61.945,161.4145,18.6787,-12112.7389
C00679=39.736,-54.260,63.612,179.7499,0.0269,-12113.7837
C00680=42.239,-58.063,65.929,-175.8220,-0.1746,-12113.9653
C00681=45.816,-62.906,68.324,-173.8645,-0.1373,-12113.9332
C00682=49.842,-68.316,70.157,-172.5980,-0.1884,-12113.8863
C00683=53.356,-73.536,71.060,-172.7432,-1.5739,-12114.0362
C00684=54.130,-79.138,71.535,-176.5613,-3.1804,-12115.6281
C00685=51.936,-84.362,71.920,-179.1729,-2.1445,-12118.3822
C00686=47.191,-88.127,72.309,-179.9965,-0.1513,-12121.8315
C00687=41.335,-91.053,72.565,179.9981,-0.0180,-12125.5835
C00688=35.156,-93.612,72.565,179.9993,-0.0181,-12129.4163
C00689=28.946,-95.684,72.309,179.9969,-0.1487,-12133.1686
C00690=22.929,-96.378,71.920,179.1719,-2.1420,-12136.6177
C00691=17.683,-94.235,71.535,176.5649,-3.1765,-12139.3722
C00692=14.270,-89.726,71.060,172.7438,-1.5775,-12140.9634
C00693=13.063,-83.550,70.157,172.5965,-0.1926,-12141.1138
C00694=12.084,-76.878,68.324,173.8594,-0.1394,-12141.0671
C00695=11.189,-70.924,65.929,175.8210,-0.1771,-12141.0349
C00696=10.270,-66.465,63.612,-179.7526,0.0255,-12141.2163
C00697=8.682,-63.886,61.945,-161.4111,18.6823,-12142.2610
C00698=5.367,-63.268,61.285,-174.0310,36.0790,-12145.1512
C00699=2.450,-63.381,61.257,179.6948,37.0092,-12147.7863
C00700=0.000,-63.425,61.276,-180.0000,37.0005,-12150.0000
C00701=-2.450,-63.381,61.257,-179.6948,37.0092,-12152.2137
C00702=-5.367,-63.268,61.285,174.0310,36.0790,-12154.8488
C00703=-8.682,-63.886,61.945,161.4119,18.6766,-12157.7390
C00704=-10.270,-66.465,63.612,179.7526,0.0255,-12158.7837
C00705=-11.189,-70.924,65.929,-175.8210,-0.1771,-12158.9651
C00706=-12.084,-76.878,68.324,-173.8594,-0.1394,-12158.9329
C00707=-13.063,-83.550,70.157,-172.5965,-0.1926,-12158.8862
C00708=-14.270,-89.726,71.060,-172.7438,-1.5775,-12159.0366
C00709=-17.683,-94.235,71.535,-176.5649,-3.1765,-12160.6278
C00710=-22.929,-96.378,71.920,-179.1719,-2.1420,-12163.3823
C00711=-28.946,-95.684,72.309,-179.9969,-0.1487,-12166.8314
C00712=-35.156,-93.612,72.565,-179.9993,-0.0181,-12170.5837
C00713=-41.335,-91.053,72.565,-179.9981,-0.0180,-12174.4165
C00714=-47.191,-88.127,72.309,179.9965,-0.1513,-12178.1685
C00715=-51.936,-84.362,71.920,179.1729,-2.1445,-12181.6178
C00716=-54.130,-79.138,71.535,176.5613,-3.1804,-12184.3719
C00717=-53.356,-73.536,71.060,172.7432,-1.5739,-12185.9638
C00718=-49.842,-68.316,70.157,172.5980,-0.1884,-12186.1137
C00719=-45.816,-62.906,68.324,173.8645,-0.1373,-12186.0668
C00720=-42.239,-58.063,65.929,175.8220,-0.1746,-12186.0347
C00721=-39.736,-54.260,63.612,-179.7499,0.0269,-12186.2163
C00722=-39.035,-51.313,61.945,-161.4145,18.6787,-12187.2611
C00723=-40.942,-48.532,61.285,-174.0315,36.0780,-12190.1513
C00724=-43.085,-46.550,61.257,179.6995,37.0101,-12192.7862
C00725=-44.848,-44.848,61.276,180.0000,36.9982,-12195.0000
C00726=-46.550,-43.085,61.257,-179.6995,37.0101,-12197.2138
C00727=-48.532,-40.942,61.285,174.0315,36.0780,-12199.8487
C00728=-51.313,-39.035,61.945,161.4145,18.6787,-12202.7389
C00729=-54.260,-39.736,63.612,179.7499,0.0269,-12203.7837
C00730=-58.063,-42.239,65.929,-175.8220,-0.1746,-12203.9653
C00731=-62.906,-45.816,68.324,-173.8645,-0.1373,-12203.9332
C00732=-68.316,-49.842,70.157,-172.5980,-0.1884,-12203.8863
C00733=-73.536,-53.356,71.060,-172.7432,-1.5739,-12204.0362
C00734=-79.138,-54.130,71.535,-176.5613,-3.1804,-12205.6281
C00735=-84.362,-51.936,71.920,-179.1729,-2.1445,-12208.3822
C00736=-88.127,-47.191,72.309,-179.9965,-0.1513,-12211.8315
C00737=-91.053,-41.335,72.565,179.9981,-0.0180,-12215.5835
C00738=-93.612,-35.156,72.565,179.9993,-0.0181,-12219.4163
C00739=-95.684,-28.946,72.309,179.9969,-0.1487,-12223.1686
C00740=-96.378,-22.929,71.920,179.1719,-2.1420,-12226.6177
C00741=-94.235,-17.683,71.535,176.5649,-3.1765,-12229.3722
C00742=-89.726,-14.270,71.060,172.7438,-1.5775,-12230.9634
C00743=-83.550,-13.063,70.157,172.5965,-0.1926,-12231.1138
C00744=-76.878,-12.084,68.324,173.8594,-0.1394,-12231.0671
C00745=-70.924,-11.189,65.929,175.8210,-0.1771,-12231.0349
C00746=-66.465,-10.270,63.612,-179.7526,0.0255,-12231.2163
C00747=-63.886,-8.682,61.945,-161.4111,18.6823,-12232.2610
C00748=-63.268,-5.367,61.285,-174.0310,36.0790,-12235.1512
C00749=-63.381,-2.450,61.257,179.6948,37.0092,-12237.7863
C00750=-63.425,0.000,61.276,180.0000,37.0005,-12240.0000
C00751=-63.381,2.450,61.257,-179.6948,37.0092,-12242.2137
C00752=-63.268,5.367,61.285,174.0310,36.0790,-12244.8488
C00753=-63.886,8.682,61.945,161.4119,18.6766,-12247.7390
C00754=-66.465,10.270,63.612,179.7526,0.0255,-12248.7837
C00755=-70.924,11.189,65.929,-175.8210,-0.1771,-12248.9651
C00756=-76.878,12.084,68.324,-173.8594,-0.1394,-12248.9329
C00757=-83.550,13.063,70.157,-172.5965,-0.1926,-12248.8862
C00758=-89.726,14.270,71.060,-172.7438,-1.5775,-12249.0366
C00759=-94.235,17.683,71.535,-176.5649,-3.1765,-12250.6278
C00760=-96.378,22.929,71.920,-179.1719,-2.1420,-12253.3823
C00761=-95.684,28.946,72.309,-179.9969,-0.1487,-12256.8314
C00762=-93.612,35.156,72.565,-179.9993,-0.0181,-12260.5837
C00763=-91.053,41.335,72.565,-179.9981,-0.0180,-12264.4165
C00764=-88.127,47.191,72.309,179.9965,-0.1513,-12268.1685
C00765=-84.362,51.936,71.920,179.1729,-2.1445,-12271.6178
C00766=-79.138,54.130,71.535,176.5613,-3.1804,-12274.3719
C00767=-73.536,53.356,71.060,172.7432,-1.5739,-12275.9638
C00768=-68.316,49.842,70.157,172.5980,-0.1884,-12276.1137
C00769=-62.906,45.816,68.324,173.8645,-0.1373,-12276.0668
C00770=-58.063,42.239,65.929,175.8220,-0.1746,-12276.0347
C00771=-54.260,39.736,63.612,-179.7499,0.0269,-12276.2163
C00772=-51.313,39.035,61.945,-161.4145,18.6787,-12277.2611
C00773=-48.532,40.942,61.285,-174.0315,36.0780,-12280.1513
C00774=-46.550,43.085,61.257,179.6995,37.0101,-12282.7862
C00775=-44.848,44.848,61.276,180.0000,36.9982,-12285.0000
C00776=-43.085,46.550,61.257,-179.6995,37.0101,-12287.2138
C00777=-40.942,48.532,61.285,174.0315,36.0780,-12289.8487
C00778=-39.035,51.313,61.945,161.4145,18.6787,-12292.7389
C00779=-39.736,54.260,63.612,179.7499,0.0269,-12293.7837
C00780=-42.239,58.063,65.929,-175.8220,-0.1746,-12293.9653
C00781=-45.816,62.906,68.324,-173.8645,-0.1373,-12293.9332
C00782=-49.842,68.316,70.157,-172.5980,-0.1884,-12293.8863
C00783=-53.356,73.536,71.060,-172.7432,-1.5739,-12294.0362
C00784=-54.130,79.138,71.535,-176.5613,-3.1804,-12295.6281
C00785=-51.936,84.362,71.920,-179.1729,-2.1445,-12298.3822
C00786=-47.191,88.127,72.309,-179.9965,-0.1513,-12301.8315
C00787=-41.335,91.053,72.565,179.9981,-0.0180,-12305.5835
C00788=-35.156,93.612,72.565,179.9993,-0.0181,-12309.4163
C00789=-28.946,95.684,72.309,179.9969,-0.1487,-12313.1686
C00790=-22.929,96.378,71.920,179.1719,-2.1420,-12316.6177
C00791=-17.683,94.235,71.535,176.5649,-3.1765,-12319.3722
C00792=-14.270,89.726,71.060,172.7438,-1.5775,-12320.9634
C00793=-13.063,83.550,70.157,172.5965,-0.1926,-12321.1138
C00794=-12.084,76.878,68.324,173.8594,-0.1394,-12321.0671
C00795=-11.189,70.924,65.929,175.8210,-0.1771,-12321.0349
C00796=-10.270,66.465,63.612,-179.7526,0.0255,-12321.2163
C00797=-8.682,63.886,61.945,-161.4119,18.6766,-12322.2610
C00798=-5.367,63.268,61.285,-174.0310,36.0790,-12325.1512
C00799=-2.450,63.381,61.257,179.6948,37.0092,-12327.7863
C00800=0.000,62.111,63.041,180.0000,36.3256,-12330.0000
C00801=2.330,62.072,63.021,-179.7028,36.3324,-12332.1497
C00802=5.165,61.970,63.050,173.8802,35.3262,-12334.7644
C00803=8.436,62.639,63.741,161.9639,17.2722,-12337.6702
C00804=9.975,65.350,65.485,-179.6415,-0.0322,-12338.6786
C00805=10.861,70.011,67.904,-175.7229,-0.1493,-12338.8182
C00806=11.743,76.212,70.393,-174.0066,-0.1107,-12338.7594
C00807=12.712,83.133,72.289,-172.8940,-0.1461,-12338.6938
C00808=13.898,89.524,73.219,-173.0501,-1.4397,-12338.8243
C00809=17.338,94.193,73.707,-176.6773,-3.0198,-12340.4296
C00810=22.659,96.427,74.103,-179.2016,-2.0437,-12343.2238
C00811=28.778,95.739,74.502,-179.9988,-0.1432,-12346.7302
C00812=35.099,93.634,74.765,-179.9993,-0.0181,-12350.5487
C00813=41.391,91.028,74.765,-179.9981,-0.0180,-12354.4516
C00814=47.349,88.047,74.502,179.9991,-0.1436,-12358.2700
C00815=52.162,84.206,74.103,179.2030,-2.0441,-12361.7764
C00816=54.344,78.865,73.707,176.6784,-3.0215,-12364.5698
C00817=53.475,73.130,73.219,173.0551,-1.4407,-12366.1755
C00818=49.795,67.773,72.289,172.8935,-0.1468,-12366.3059
C00819=45.586,62.194,70.393,174.0079,-0.1079,-12366.2401
C00820=41.825,57.185,67.904,175.7207,-0.1531,-12366.1817
C00821=39.156,53.262,65.485,179.6421,-0.0355,-12366.3218
C00822=38.328,50.258,63.741,-161.9596,17.2759,-12367.3300
C00823=40.167,47.472,63.050,-173.8825,35.3269,-12370.2352
C00824=42.244,45.539,63.021,179.7046,36.3332,-12372.8504
C00825=43.919,43.919,63.041,-180.0000,36.3263,-12375.0000
C00826=45.539,42.244,63.021,-179.7046,36.3332,-12377.1496
C00827=47.472,40.167,63.050,173.8780,35.3233,-12379.7648
C00828=50.258,38.328,63.741,161.9596,17.2759,-12382.6700
C00829=53.262,39.156,65.485,-179.6421,-0.0355,-12383.6782
C00830=57.185,41.825,67.904,-175.7207,-0.1531,-12383.8183
C00831=62.194,45.586,70.393,-174.0079,-0.1079,-12383.7599
C00832=67.773,49.795,72.289,-172.8935,-0.1468,-12383.6941
C00833=73.130,53.475,73.219,-173.0551,-1.4407,-12383.8245
C00834=78.865,54.344,73.707,-176.6784,-3.0215,-12385.4302
C00835=84.206,52.162,74.103,-179.2030,-2.0441,-12388.2236
C00836=88.047,47.349,74.502,-179.9991,-0.1436,-12391.7300
C00837=91.028,41.391,74.765,179.9981,-0.0180,-12395.5484
C00838=93.634,35.099,74.765,179.9993,-0.0181,-12399.4513
C00839=95.739,28.778,74.502,179.9988,-0.1432,-12403.2698
C00840=96.427,22.659,74.103,179.2016,-2.0437,-12406.7762
C00841=94.193,17.338,73.707,176.6773,-3.0198,-12409.5704
C00842=89.524,13.898,73.219,173.0501,-1.4397,-12411.1757
C00843=83.133,12.712,72.289,172.8940,-0.1461,-12411.3062
C00844=76.212,11.743,70.393,174.0066,-0.1107,-12411.2406
C00845=70.011,10.861,67.904,175.7229,-0.1493,-12411.1818
C00846=65.350,9.975,65.485,179.6415,-0.0322,-12411.3214
C00847=62.639,8.436,63.741,-161.9639,17.2722,-12412.3298
C00848=61.970,5.165,63.050,-173.8802,35.3262,-12415.2356
C00849=62.072,2.330,63.021,179.7028,36.3324,-12417.8503
C00850=62.111,0.000,63.041,-180.0000,36.3256,-12420.0000
C00851=62.072,-2.330,63.021,-179.7028,36.3324,-12422.1497
C00852=61.970,-5.165,63.050,173.8802,35.3262,-12424.7644
C00853=62.640,-8.436,63.741,161.9639,17.2723,-12427.6701
C00854=65.350,-9.975,65.485,-179.6415,-0.0322,-12428.6786
C00855=70.011,-10.861,67.904,-175.7229,-0.1493,-12428.8182
C00856=76.212,-11.743,70.393,-174.0066,-0.1107,-12428.7594
C00857=83.133,-12.712,72.289,-172.8940,-0.1461,-12428.6938
C00858=89.524,-13.898,73.219,-173.0501,-1.4397,-12428.8243
C00859=94.193,-17.338,73.707,-176.6773,-3.0198,-12430.4296
C00860=96.427,-22.659,74.103,-179.2016,-2.0437,-12433.2238
C00861=95.739,-28.778,74.502,-179.9988,-0.1432,-12436.7302
C00862=93.634,-35.099,74.765,-179.9993,-0.0181,-12440.5487
C00863=91.028,-41.391,74.765,-179.9981,-0.0180,-12444.4516
C00864=88.047,-47.349,74.502,179.9991,-0.1436,-12448.2700
C00865=84.206,-52.162,74.103,179.2030,-2.0441,-12451.7764
C00866=78.865,-54.344,73.707,176.6784,-3.0215,-12454.5698
C00867=73.130,-53.475,73.219,173.0551,-1.4407,-12456.1755
C00868=67.773,-49.795,72.289,172.8935,-0.1468,-12456.3059
C00869=62.194,-45.586,70.393,174.0079,-0.1079,-12456.2401
C00870=57.185,-41.825,67.904,175.7207,-0.1531,-12456.1817
C00871=53.262,-39.156,65.485,179.6421,-0.0355,-12456.3218
C00872=50.258,-38.328,63.741,-161.9596,17.2759,-12457.3300
C00873=47.472,-40.167,63.050,-173.8825,35.3269,-12460.2352
C00874=45.539,-42.244,63.021,179.7046,36.3332,-12462.8504
C00875=43.919,-43.919,63.041,-180.0000,36.3263,-12465.0000
C00876=42.244,-45.539,63.021,-179.7046,36.3332,-12467.1496
C00877=40.167,-47.472,63.050,173.8780,35.3233,-12469.7648
C00878=38.328,-50.258,63.741,161.9596,17.2759,-12472.6700
C00879=39.156,-53.262,65.485,-179.6421,-0.0355,-12473.6782
C00880=41.825,-57.185,67.904,-175.7207,-0.1531,-12473.8183
C00881=45.586,-62.194,70.393,-174.0079,-0.1079,-12473.7599
C00882=49.795,-67.773,72.289,-172.8935,-0.1468,-12473.6941
C00883=53.475,-73.130,73.219,-173.0551,-1.4407,-12473.8245
C00884=54.344,-78.865,73.707,-176.6784,-3.0215,-12475.4302
C00885=52.162,-84.206,74.103,-179.2030,-2.0441,-12478.2236
C00886=47.349,-88.047,74.502,-179.9991,-0.1436,-12481.7300
C00887=41.391,-91.028,74.765,179.9981,-0.0180,-12485.5484
C00888=35.099,-93.634,74.765,179.9993,-0.0181,-12489.4513
C00889=28.778,-95.739,74.502,179.9988,-0.1432,-12493.2698
C00890=22.659,-96.427,74.103,179.2016,-2.0437,-12496.7762
C00891=17.338,-94.193,73.707,176.6773,-3.0198,-12499.5704
C00892=13.898,-89.524,73.219,173.0501,-1.4397,-12501.1757
C00893=12.712,-83.133,72.289,172.8940,-0.1461,-12501.3062
C00894=11.743,-76.212,70.393,174.0066,-0.1107,-12501.2406
C00895=10.861,-70.011,67.904,175.7229,-0.1493,-12501.1818
C00896=9.975,-65.350,65.485,179.6415,-0.0322,-12501.3214
C00897=8.436,-62.639,63.741,-161.9639,17.2722,-12502.3298
C00898=5.165,-61.970,63.050,-173.8802,35.3262,-12505.2356
C00899=2.330,-62.072,63.021,179.7028,36.3324,-12507.8503
C00900=0.000,-62.111,63.041,-180.0000,36.3256,-12510.0000
C00901=-2.330,-62.072,63.021,-179.7028,36.3324,-12512.1497
C00902=-5.165,-61.970,63.050,173.8802,35.3262,-12514.7644
C00903=-8.436,-62.640,63.741,161.9639,17.2723,-12517.6701
C00904=-9.975,-65.350,65.485,-179.6415,-0.0322,-12518.6786
C00905=-10.861,-70.011,67.904,-175.7229,-0.1493,-12518.8182
C00906=-11.743,-76.212,70.393,-174.0066,-0.1107,-12518.7594
C00907=-12.712,-83.133,72.289,-172.8940,-0.1461,-12518.6938
C00908=-13.898,-89.524,73.219,-173.0501,-1.4397,-12518.8243
C00909=-17.338,-94.193,73.707,-176.6773,-3.0198,-12520.4296
C00910=-22.659,-96.427,74.103,-179.2016,-2.0437,-12523.2238
C00911=-28.778,-95.739,74.502,-179.9988,-0.1432,-12526.7302
C00912=-35.099,-93.634,74.765,-179.9993,-0.0181,-12530.5487
C00913=-41.391,-91.028,74.765,-179.9981,-0.0180,-12534.4516
C00914=-47.349,-88.047,74.502,179.9991,-0.1436,-12538.2700
C00915=-52.162,-84.206,74.103,179.2030,-2.0441,-12541.7764
C00916=-54.344,-78.865,73.707,176.6784,-3.0215,-12544.5698
C00917=-53.475,-73.130,73.219,173.0551,-1.4407,-12546.1755
C00918=-49.795,-67.773,72.289,172.8935,-0.1468,-12546.3059
C00919=-45.586,-62.194,70.393,174.0079,-0.1079,-12546.2401
C00920=-41.825,-57.185,67.904,175.7207,-0.1531,-12546.1817
C00921=-39.156,-53.262,65.485,179.6421,-0.0355,-12546.3218
C00922=-38.328,-50.258,63.741,-161.9596,17.2759,-12547.3300
C00923=-40.167,-47.472,63.050,-173.8825,35.3269,-12550.2352
C00924=-42.244,-45.539,63.021,179.7046,36.3332,-12552.8504
C00925=-43.919,-43.919,63.041,-180.0000,36.3263,-12555.0000
C00926=-45.539,-42.244,63.021,-179.7046,36.3332,-12557.1496
C00927=-47.472,-40.167,63.050,173.8780,35.3233,-12559.7648
C00928=-50.258,-38.328,63.741,161.9596,17.2759,-12562.6700
C00929=-53.262,-39.156,65.485,-179.6421,-0.0355,-12563.6782
C00930=-57.185,-41.825,67.904,-175.7207,-0.1531,-12563.8183
C00931=-62.194,-45.586,70.393,-174.0079,-0.1079,-12563.7599
C00932=-67.773,-49.795,72.289,-172.8935,-0.1468,-12563.6941
C00933=-73.130,-53.475,73.219,-173.0551,-1.4407,-12563.8245
C00934=-78.865,-54.344,73.707,-176.6784,-3.0215,-12565.4302
C00935=-84.206,-52.162,74.103,-179.2030,-2.0441,-12568.2236
C00936=-88.047,-47.349,74.502,-179.9991,-0.1436,-12571.7300
C00937=-91.028,-41.391,74.765,179.9981,-0.0180,-12575.5484
C00938=-93.634,-35.099,74.765,179.9993,-0.0181,-12579.4513
C00939=-95.739,-28.778,74.502,179.9988,-0.1432,-12583.2698
C00940=-96.427,-22.659,74.103,179.2016,-2.0437,-12586.7762
C00941=-94.193,-17.338,73.707,176.6773,-3.0198,-12589.5704
C00942=-89.524,-13.898,73.219,173.0501,-1.4397,-12591.1757
C00943=-83.133,-12.712,72.289,172.8940,-0.1461,-12591.3062
C00944=-76.212,-11.743,70.393,174.0066,-0.1107,-12591.2406
C00945=-70.011,-10.861,67.904,175.7229,-0.1493,-12591.1818
C00946=-65.350,-9.975,65.485,179.6415,-0.0322,-12591.3214
C00947=-62.639,-8.436,63.741,-161.9639,17.2722,-12592.3298
C00948=-61.970,-5.165,63.050,-173.8802,35.3262,-12595.2356
C00949=-62.072,-2.330,63.021,179.7028,36.3324,-12597.8503
C00950=-62.111,0.000,63.041,-180.0000,36.3256,-12600.0000
C00951=-62.072,2.330,63.021,-179.7028,36.3324,-12602.1497
C00952=-61.970,5.165,63.050,173.8802,35.3262,-12604.7644
C00953=-62.640,8.436,63.741,161.9639,17.2723,-12607.6701
C00954=-65.350,9.975,65.485,-179.6415,-0.0322,-12608.6786
C00955=-70.011,10.861,67.904,-175.7229,-0.1493,-12608.8182
C00956=-76.212,11.743,70.393,-174.0066,-0.1107,-12608.7594
C00957=-83.133,12.712,72.289,-172.8940,-0.1461,-12608.6938
C00958=-89.524,13.898,73.219,-173.0501,-1.4397,-12608.8243
C00959=-94.193,17.338,73.707,-176.6773,-3.0198,-12610.4296
C00960=-96.427,22.659,74.103,-179.2016,-2.0437,-12613.2238
C00961=-95.739,28.778,74.502,-179.9988,-0.1432,-12616.7302
C00962=-93.634,35.099,74.765,-179.9993,-0.0181,-12620.5487
C00963=-91.028,41.391,74.765,-179.9981,-0.0180,-12624.4516
C00964=-88.047,47.349,74.502,179.9991,-0.1436,-12628.2700
C00965=-84.206,52.162,74.103,179.2030,-2.0441,-12631.7764
C00966=-78.865,54.344,73.707,176.6784,-3.0215,-12634.5698
C00967=-73.130,53.475,73.219,173.0551,-1.4407,-12636.1755
C00968=-67.773,49.795,72.289,172.8935,-0.1468,-12636.3059
C00969=-62.194,45.586,70.393,174.0079,-0.1079,-12636.2401
C00970=-57.185,41.825,67.904,175.7207,-0.1531,-12636.1817
C00971=-53.262,39.156,65.485,179.6421,-0.0355,-12636.3218
C00972=-50.258,38.328,63.741,-161.9596,17.2759,-12637.3300
C00973=-47.472,40.167,63.050,-173.8825,35.3269,-12640.2352
C00974=-45.539,42.244,63.021,179.7046,36.3332,-12642.8504
C00975=-43.919,43.919,63.041,180.0000,36.3263,-12645.0000
C00976=-42.244,45.539,63.021,-179.7046,36.3332,-12647.1496
C00977=-40.167,47.472,63.050,173.8780,35.3233,-12649.7648
C00978=-38.328,50.258,63.741,161.9596,17.2759,-12652.6700
C00979=-39.156,53.262,65.485,-179.6421,-0.0355,-12653.6782
C00980=-41.825,57.185,67.904,-175.7207,-0.1531,-12653.8183
C00981=-45.586,62.194,70.393,-174.0079,-0.1079,-12653.7599
C00982=-49.795,67.773,72.289,-172.8935,-0.1468,-12653.6941
C00983=-53.475,73.130,73.219,-173.0551,-1.4407,-12653.8245
C00984=-54.344,78.865,73.707,-176.6784,-3.0215,-12655.4302
C00985=-52.162,84.206,74.103,-179.2030,-2.0441,-12658.2236
C00986=-47.349,88.047,74.502,-179.9991,-0.1436,-12661.7300
C00987=-41.391,91.028,74.765,179.9981,-0.0180,-12665.5484
C00988=-35.099,93.634,74.765,179.9993,-0.0181,-12669.4513
C00989=-28.778,95.739,74.502,179.9988,-0.1432,-12673.2698
C00990=-22.659,96.427,74.103,179.2016,-2.0437,-12676.7762
C00991=-17.338,94.193,73.707,176.6773,-3.0198,-12679.5704
C00992=-13.898,89.524,73.219,173.0501,-1.4397,-12681.1757
C00993=-12.712,83.133,72.289,172.8940,-0.1461,-12681.3062
C00994=-11.743,76.212,70.393,174.0066,-0.1107,-12681.2406
C00995=-10.861,70.011,67.904,175.7229,-0.1493,-12681.1818
C00996=-9.975,65.350,65.485,179.6415,-0.0322,-12681.3214
C00997=-8.436,62.640,63.741,-161.9639,17.2723,-12682.3299
C00998=-5.165,61.970,63.050,-173.8802,35.3262,-12685.2356
C00999=-2.330,62.072,63.021,179.7028,36.3324,-12687.8503
C01000=0.000,60.820,64.822,180.0000,35.5497,-12690.0000
C01001=2.212,60.785,64.801,-179.7074,35.5593,-12692.0841
C01002=4.967,60.695,64.832,173.7605,34.4682,-12694.6784
C01003=8.195,61.417,65.554,162.6105,15.8904,-12697.6002
C01004=9.686,64.262,67.375,-179.1259,-0.0711,-12698.5715
C01005=10.544,69.129,69.894,-175.6880,-0.1257,-12698.6723
C01006=11.418,75.576,72.474,-174.2120,-0.0836,-12698.5913
C01007=12.382,82.740,74.428,-173.2591,-0.1124,-12698.5111
C01008=13.550,89.334,75.383,-173.4296,-1.3094,-12698.6248
C01009=17.016,94.154,75.883,-176.8342,-2.8344,-12700.2442
C01010=22.407,96.473,76.288,-179.2397,-1.9299,-12703.0758
C01011=28.621,95.791,76.696,179.9993,-0.1377,-12706.6354
C01012=35.046,93.654,76.964,-179.9993,-0.0181,-12710.5162
C01013=41.442,91.005,76.964,-179.9981,-0.0180,-12714.4836
C01014=47.497,87.973,76.696,-179.9983,-0.1358,-12718.3648
C01015=52.372,84.060,76.288,179.2407,-1.9248,-12721.9242
C01016=54.545,78.609,75.883,176.8367,-2.8312,-12724.7559
C01017=53.588,72.750,75.383,173.4272,-1.3089,-12726.3755
C01018=49.751,67.261,74.428,173.2583,-0.1085,-12726.4893
C01019=45.367,61.514,72.474,174.2127,-0.0823,-12726.4090
C01020=41.426,56.337,69.894,175.6860,-0.1257,-12726.3280
C01021=38.591,52.289,67.375,179.1285,-0.0735,-12726.4285
C01022=37.634,49.223,65.554,-162.6128,15.8893,-12727.4001
C01023=39.406,46.429,64.832,-173.7617,34.4707,-12730.3225
C01024=41.417,44.545,64.801,179.7113,35.5606,-12732.9160
C01025=43.006,43.006,64.822,180.0000,35.5489,-12735.0000
C01026=44.545,41.417,64.801,-179.7113,35.5606,-12737.0840
C01027=46.430,39.405,64.832,173.7564,34.4670,-12739.6788
C01028=49.223,37.634,65.554,162.6128,15.8893,-12742.5999
C01029=52.289,38.591,67.375,-179.1285,-0.0735,-12743.5715
C01030=56.337,41.426,69.894,-175.6860,-0.1257,-12743.6720
C01031=61.514,45.367,72.474,-174.2127,-0.0823,-12743.5910
C01032=67.261,49.751,74.428,-173.2583,-0.1085,-12743.5107
C01033=72.750,53.588,75.383,-173.4272,-1.3089,-12743.6245
C01034=78.609,54.545,75.883,-176.8367,-2.8312,-12745.2441
C01035=84.060,52.372,76.288,-179.2407,-1.9248,-12748.0758
C01036=87.973,47.497,76.696,179.9983,-0.1358,-12751.6352
C01037=91.005,41.442,76.964,179.9981,-0.0180,-12755.5164
C01038=93.654,35.046,76.964,179.9993,-0.0181,-12759.4838
C01039=95.791,28.621,76.696,-179.9993,-0.1377,-12763.3646
C01040=96.473,22.407,76.288,179.2397,-1.9299,-12766.9242
C01041=94.154,17.016,75.883,176.8342,-2.8344,-12769.7558
C01042=89.334,13.550,75.383,173.4296,-1.3094,-12771.3752
C01043=82.740,12.382,74.428,173.2591,-0.1124,-12771.4889
C01044=75.576,11.418,72.474,174.2120,-0.0836,-12771.4087
C01045=69.129,10.544,69.894,175.6880,-0.1257,-12771.3277
C01046=64.262,9.686,67.375,179.1259,-0.0711,-12771.4285
C01047=61.417,8.195,65.554,-162.6105,15.8904,-12772.3998
C01048=60.695,4.967,64.832,-173.7605,34.4682,-12775.3216
C01049=60.785,2.212,64.801,179.7074,35.5593,-12777.9159
C01050=60.820,0.000,64.822,180.0000,35.5497,-12780.0000
C01051=60.785,-2.212,64.801,-179.7074,35.5593,-12782.0841
C01052=60.695,-4.967,64.832,173.7605,34.4682,-12784.6784
C01053=61.417,-8.195,65.554,162.6105,15.8904,-12787.6002
C01054=64.262,-9.686,67.375,-179.1259,-0.0711,-12788.5715
C01055=69.129,-10.544,69.894,-175.6880,-0.1257,-12788.6723
C01056=75.576,-11.418,72.474,-174.2120,-0.0836,-12788.5913
C01057=82.740,-12.382,74.428,-173.2591,-0.1124,-12788.5111
C01058=89.334,-13.550,75.383,-173.4296,-1.3094,-12788.6248
C01059=94.154,-17.016,75.883,-176.8342,-2.8344,-12790.2442
C01060=96.473,-22.407,76.288,-179.2397,-1.9299,-12793.0758
C01061=95.791,-28.621,76.696,179.9993,-0.1377,-12796.6354
C01062=93.654,-35.046,76.964,-179.9993,-0.0181,-12800.5162
C01063=91.005,-41.442,76.964,-179.9981,-0.0180,-12804.4836
C01064=87.973,-47.497,76.696,-179.9983,-0.1358,-12808.3648
C01065=84.060,-52.372,76.288,179.2407,-1.9248,-12811.9242
C01066=78.609,-54.545,75.883,176.8367,-2.8312,-12814.7559
C01067=72.750,-53.588,75.383,173.4272,-1.3089,-12816.3755
C01068=67.261,-49.751,74.428,173.2583,-0.1085,-12816.4893
C01069=61.514,-45.367,72.474,174.2127,-0.0823,-12816.4090
C01070=56.337,-41.426,69.894,175.6860,-0.1257,-12816.3280
C01071=52.289,-38.591,67.375,179.1285,-0.0735,-12816.4285
C01072=49.223,-37.634,65.554,-162.6128,15.8893,-12817.4001
C01073=46.429,-39.406,64.832,-173.7617,34.4707,-12820.3225
C01074=44.545,-41.417,64.801,179.7113,35.5606,-12822.9160
C01075=43.006,-43.006,64.822,-180.0000,35.5489,-12825.0000
C01076=41.417,-44.545,64.801,-179.7113,35.5606,-12827.0840
C01077=39.405,-46.430,64.832,173.7564,34.4670,-12829.6788
C01078=37.634,-49.223,65.554,162.6128,15.8893,-12832.5999
C01079=38.591,-52.289,67.375,-179.1285,-0.0735,-12833.5715
C01080=41.426,-56.337,69.894,-175.6860,-0.1257,-12833.6720
C01081=45.367,-61.514,72.474,-174.2127,-0.0823,-12833.5910
C01082=49.751,-67.261,74.428,-173.2583,-0.1085,-12833.5107
C01083=53.588,-72.750,75.383,-173.4272,-1.3089,-12833.6245
C01084=54.545,-78.609,75.883,-176.8367,-2.8312,-12835.2441
C01085=52.372,-84.060,76.288,-179.2407,-1.9248,-12838.0758
C01086=47.497,-87.973,76.696,179.9983,-0.1358,-12841.6352
C01087=41.442,-91.005,76.964,179.9981,-0.0180,-12845.5164
C01088=35.046,-93.654,76.964,179.9993,-0.0181,-12849.4838
C01089=28.621,-95.791,76.696,-179.9993,-0.1377,-12853.3646
C01090=22.407,-96.473,76.288,179.2397,-1.9299,-12856.9242
C01091=17.016,-94.154,75.883,176.8342,-2.8344,-12859.7558
C01092=13.550,-89.334,75.383,173.4296,-1.3094,-12861.3752
C01093=12.382,-82.740,74.428,173.2591,-0.1124,-12861.4889
C01094=11.418,-75.576,72.474,174.2120,-0.0836,-12861.4087
C01095=10.544,-69.129,69.894,175.6880,-0.1257,-12861.3277
C01096=9.686,-64.262,67.375,179.1259,-0.0711,-12861.4285
C01097=8.195,-61.417,65.554,-162.6105,15.8904,-12862.3998
C01098=4.967,-60.695,64.832,-173.7605,34.4682,-12865.3216
C01099=2.212,-60.785,64.801,179.7074,35.5593,-12867.9159
C01100=0.000,-60.820,64.822,-180.0000,35.5497,-12870.0000
C01101=-2.212,-60.785,64.801,-179.7074,35.5593,-12872.0841
C01102=-4.967,-60.695,64.832,173.7605,34.4682,-12874.6784
C01103=-8.195,-61.417,65.554,162.6105,15.8904,-12877.6002
C01104=-9.686,-64.262,67.375,-179.1259,-0.0711,-12878.5715
C01105=-10.544,-69.129,69.894,-175.6880,-0.1257,-12878.6723
C01106=-11.418,-75.576,72.474,-174.2120,-0.0836,-12878.5913
C01107=-12.382,-82.740,74.428,-173.2591,-0.1124,-12878.5111
C01108=-13.550,-89.334,75.383,-173.4296,-1.3094,-12878.6248
C01109=-17.016,-94.154,75.883,-176.8342,-2.8344,-12880.2442
C01110=-22.407,-96.473,76.288,-179.2397,-1.9299,-12883.0758
C01111=-28.621,-95.791,76.696,179.9993,-0.1377,-12886.6354
C01112=-35.046,-93.654,76.964,-179.9993,-0.0181,-12890.5162
C01113=-41.442,-91.005,76.964,-179.9981,-0.0180,-12894.4836
C01114=-47.497,-87.973,76.696,-179.9983,-0.1358,-12898.3648
C01115=-52.372,-84.060,76.288,179.2407,-1.9248,-12901.9242
C01116=-54.545,-78.609,75.883,176.8367,-2.8312,-12904.7559
C01117=-53.588,-72.750,75.383,173.4272,-1.3089,-12906.3755
C01118=-49.751,-67.261,74.428,173.2583,-0.1085,-12906.4893
C01119=-45.367,-61.514,72.474,174.2127,-0.0823,-12906.4090
C01120=-41.426,-56.337,69.894,175.6860,-0.1257,-12906.3280
C01121=-38.591,-52.289,67.375,179.1285,-0.0735,-12906.4285
C01122=-37.634,-49.223,65.554,-162.6128,15.8893,-12907.4001
C01123=-39.406,-46.429,64.832,-173.7617,34.4707,-12910.3225
C01124=-41.417,-44.545,64.801,179.7113,35.5606,-12912.9160
C01125=-43.006,-43.006,64.822,-180.0000,35.5489,-12915.0000
C01126=-44.545,-41.417,64.801,-179.7113,35.5606,-12917.0840
C01127=-46.430,-39.405,64.832,173.7564,34.4670,-12919.6788
C01128=-49.223,-37.634,65.554,162.6128,15.8893,-12922.5999
C01129=-52.289,-38.591,67.375,-179.1285,-0.0735,-12923.5715
C01130=-56.337,-41.426,69.894,-175.6860,-0.1257,-12923.6720
C01131=-61.514,-45.367,72.474,-174.2127,-0.0823,-12923.5910
C01132=-67.261,-49.751,74.428,-173.2583,-0.1085,-12923.5107
C01133=-72.750,-53.588,75.383,-173.4272,-1.3089,-12923.6245
C01134=-78.609,-54.545,75.883,-176.8367,-2.8312,-12925.2441
C01135=-84.060,-52.372,76.288,-179.2407,-1.9248,-12928.0758
C01136=-87.973,-47.497,76.696,179.9983,-0.1358,-12931.6352
C01137=-91.005,-41.442,76.964,179.9981,-0.0180,-12935.5164
C01138=-93.654,-35.046,76.964,179.9993,-0.0181,-12939.4838
C01139=-95.791,-28.621,76.696,-179.9993,-0.1377,-12943.3646
C01140=-96.473,-22.407,76.288,179.2397,-1.9299,-12946.9242
C01141=-94.154,-17.016,75.883,176.8342,-2.8344,-12949.7558
C01142=-89.334,-13.550,75.383,173.4296,-1.3094,-12951.3752
C01143=-82.740,-12.382,74.428,173.2591,-0.1124,-12951.4889
C01144=-75.576,-11.418,72.474,174.2120,-0.0836,-12951.4087
C01145=-69.129,-10.544,69.894,175.6880,-0.1257,-12951.3277
C01146=-64.262,-9.686,67.375,179.1259,-0.0711,-12951.4285
C01147=-61.417,-8.195,65.554,-162.6105,15.8904,-12952.3998
C01148=-60.695,-4.967,64.832,-173.7605,34.4682,-12955.3216
C01149=-60.785,-2.212,64.801,179.7074,35.5593,-12957.9159
C01150=-60.820,0.000,64.822,-180.0000,35.5497,-12960.0000
C01151=-60.785,2.212,64.801,-179.7074,35.5593,-12962.0841
C01152=-60.695,4.967,64.832,173.7605,34.4682,-12964.6784
C01153=-61.417,8.195,65.554,162.6105,15.8904,-12967.6002
C01154=-64.262,9.686,67.375,-179.1259,-0.0711,-12968.5715
C01155=-69.129,10.544,69.894,-175.6880,-0.1257,-12968.6723
C01156=-75.576,11.418,72.474,-174.2120,-0.0836,-12968.5913
C01157=-82.740,12.382,74.428,-173.2591,-0.1124,-12968.5111
C01158=-89.334,13.550,75.383,-173.4296,-1.3094,-12968.6248
C01159=-94.154,17.016,75.883,-176.8342,-2.8344,-12970.2442
C01160=-96.473,22.407,76.288,-179.2397,-1.9299,-12973.0758
C01161=-95.791,28.621,76.696,179.9993,-0.1377,-12976.6354
C01162=-93.654,35.046,76.964,-179.9993,-0.0181,-12980.5162
C01163=-91.005,41.442,76.964,-179.9981,-0.0180,-12984.4836
C01164=-87.973,47.497,76.696,-179.9983,-0.1358,-12988.3648
C01165=-84.060,52.372,76.288,179.2407,-1.9248,-12991.9242
C01166=-78.609,54.545,75.883,176.8367,-2.8312,-12994.7559
C01167=-72.750,53.588,75.383,173.4272,-1.3089,-12996.3755
C01168=-67.261,49.751,74.428,173.2583,-0.1085,-12996.4893
C01169=-61.514,45.367,72.474,174.2127,-0.0823,-12996.4090
C01170=-56.337,41.426,69.894,175.6860,-0.1257,-12996.3280
C01171=-52.289,38.591,67.375,179.1285,-0.0735,-12996.4285
C01172=-49.223,37.634,65.554,-162.6128,15.8893,-12997.4001
C01173=-46.429,39.406,64.832,-173.7617,34.4707,-13000.3225
C01174=-44.545,41.417,64.801,179.7113,35.5606,-13002.9160
C01175=-43.006,43.006,64.822,-180.0000,35.5489,-13005.0000
C01176=-41.417,44.545,64.801,-179.7113,35.5606,-13007.0840
C01177=-39.405,46.430,64.832,173.7564,34.4670,-13009.6788
C01178=-37.634,49.223,65.554,162.6128,15.8893,-13012.5999
C01179=-38.591,52.289,67.375,-179.1285,-0.0735,-13013.5715
C01180=-41.426,56.337,69.894,-175.6860,-0.1257,-13013.6720
C01181=-45.367,61.514,72.474,-174.2127,-0.0823,-13013.5910
C01182=-49.751,67.261,74.428,-173.2583,-0.1085,-13013.5107
C01183=-53.588,72.750,75.383,-173.4272,-1.3089,-13013.6245
C01184=-54.545,78.609,75.883,-176.8367,-2.8312,-13015.2441
C01185=-52.372,84.060,76.288,-179.2407,-1.9248,-13018.0758
C01186=-47.497,87.973,76.696,179.9983,-0.1358,-13021.6352
C01187=-41.442,91.005,76.964,179.9981,-0.0180,-13025.5164
C01188=-35.046,93.654,76.964,179.9993,-0.0181,-13029.4838
C01189=-28.621,95.791,76.696,-179.9993,-0.1377,-13033.3646
C01190=-22.407,96.473,76.288,179.2397,-1.9299,-13036.9242
C01191=-17.016,94.154,75.883,176.8342,-2.8344,-13039.7558
C01192=-13.550,89.334,75.383,173.4296,-1.3094,-13041.3752
C01193=-12.382,82.740,74.428,173.2591,-0.1124,-13041.4889
C01194=-11.418,75.576,72.474,174.2120,-0.0836,-13041.4087
C01195=-10.544,69.129,69.894,175.6880,-0.1257,-13041.3277
C01196=-9.686,64.262,67.375,179.1259,-0.0711,-13041.4285
C01197=-8.195,61.417,65.554,-162.6105,15.8904,-13042.3998
C01198=-4.967,60.695,64.832,-173.7605,34.4682,-13045.3216
C01199=-2.212,60.785,64.801,179.7074,35.5593,-13047.9159
C01200=0.000,59.554,66.621,-180.0000,34.6578,-13050.0000
C01201=2.097,59.523,66.599,-179.7230,34.6655,-13052.0177
C01202=4.772,59.445,66.632,173.6798,33.4987,-13054.5896
C01203=7.959,60.221,67.386,163.3494,14.5335,-13057.5288
C01204=9.406,63.206,69.285,-178.7004,-0.0905,-13058.4644
C01205=10.239,68.282,71.901,-175.7112,-0.0994,-13058.5281
C01206=11.109,74.974,74.567,-174.4741,-0.0631,-13058.4283
C01207=12.073,82.372,76.575,-173.6811,-0.0780,-13058.3383
C01208=13.226,89.158,77.551,-173.8761,-1.1797,-13058.4379
C01209=16.717,94.118,78.062,-177.0287,-2.6199,-13060.0717
C01210=22.174,96.515,78.476,-179.2889,-1.7890,-13062.9390
C01211=28.477,95.839,78.891,-179.9987,-0.1251,-13066.5485
C01212=34.998,93.673,79.163,179.9986,-0.0127,-13070.4866
C01213=41.489,90.984,79.163,179.9995,-0.0128,-13074.5131
C01214=47.632,87.904,78.891,179.9965,-0.1257,-13078.4517
C01215=52.567,83.926,78.476,179.2889,-1.7910,-13082.0609
C01216=54.731,78.373,78.062,177.0289,-2.6213,-13084.9281
C01217=53.692,72.396,77.551,173.8708,-1.1760,-13086.5622
C01218=49.709,66.782,76.575,173.6819,-0.0796,-13086.6621
C01219=45.159,60.870,74.567,174.4737,-0.0632,-13086.5714
C01220=41.042,55.523,71.901,175.7117,-0.1034,-13086.4714
C01221=38.042,51.344,69.285,178.6998,-0.0933,-13086.5356
C01222=36.955,48.211,67.386,-163.3536,14.5351,-13087.4711
C01223=38.660,45.408,66.632,-173.6783,33.4962,-13090.4108
C01224=40.607,43.572,66.599,179.7247,34.6655,-13092.9827
C01225=42.111,42.111,66.621,-180.0000,34.6557,-13095.0000
C01226=43.571,40.607,66.599,-179.7195,34.6689,-13097.0166
C01227=45.409,38.659,66.632,173.6775,33.4961,-13099.5906
C01228=48.211,36.955,67.386,163.3501,14.5305,-13102.5289
C01229=51.344,38.042,69.285,-178.6998,-0.0933,-13103.4644
C01230=55.523,41.042,71.901,-175.7117,-0.1034,-13103.5286
C01231=60.870,45.159,74.567,-174.4737,-0.0632,-13103.4286
C01232=66.782,49.709,76.575,-173.6819,-0.0796,-13103.3379
C01233=72.396,53.692,77.551,-173.8708,-1.1760,-13103.4378
C01234=78.373,54.731,78.062,-177.0289,-2.6213,-13105.0719
C01235=83.926,52.567,78.476,-179.2889,-1.7910,-13107.9391
C01236=87.904,47.632,78.891,-179.9965,-0.1257,-13111.5483
C01237=90.984,41.489,79.163,-179.9995,-0.0128,-13115.4869
C01238=93.673,34.998,79.163,-179.9986,-0.0127,-13119.5134
C01239=95.839,28.477,78.891,179.9987,-0.1251,-13123.4515
C01240=96.515,22.174,78.476,179.2889,-1.7890,-13127.0610
C01241=94.118,16.717,78.062,177.0287,-2.6199,-13129.9283
C01242=89.158,13.226,77.551,173.8761,-1.1797,-13131.5621
C01243=82.372,12.073,76.575,173.6811,-0.0780,-13131.6617
C01244=74.974,11.109,74.567,174.4741,-0.0631,-13131.5717
C01245=68.282,10.239,71.901,175.7112,-0.0994,-13131.4719
C01246=63.206,9.406,69.285,178.7004,-0.0905,-13131.5356
C01247=60.221,7.959,67.386,-163.3494,14.5335,-13132.4712
C01248=59.445,4.772,66.632,-173.6798,33.4987,-13135.4104
C01249=59.523,2.097,66.599,179.7230,34.6655,-13137.9823
C01250=59.554,0.000,66.621,180.0000,34.6578,-13140.0000
C01251=59.523,-2.096,66.599,-179.7223,34.6655,-13142.0167
C01252=59.445,-4.772,66.632,173.6803,33.4939,-13144.5896
C01253=60.222,-7.959,67.386,163.3494,14.5335,-13147.5286
C01254=63.206,-9.406,69.285,-178.7004,-0.0905,-13148.4644
C01255=68.282,-10.239,71.901,-175.7112,-0.0994,-13148.5281
C01256=74.974,-11.109,74.567,-174.4741,-0.0631,-13148.4283
C01257=82.372,-12.073,76.575,-173.6811,-0.0780,-13148.3383
C01258=89.158,-13.226,77.551,-173.8761,-1.1797,-13148.4379
C01259=94.118,-16.717,78.062,-177.0287,-2.6199,-13150.0717
C01260=96.515,-22.174,78.476,-179.2889,-1.7890,-13152.9390
C01261=95.839,-28.477,78.891,-179.9987,-0.1251,-13156.5485
C01262=93.673,-34.998,79.163,179.9986,-0.0127,-13160.4866
C01263=90.984,-41.489,79.163,179.9995,-0.0128,-13164.5131
C01264=87.904,-47.632,78.891,179.9965,-0.1257,-13168.4517
C01265=83.926,-52.567,78.476,179.2889,-1.7910,-13172.0609
C01266=78.373,-54.731,78.062,177.0289,-2.6213,-13174.9281
C01267=72.396,-53.692,77.551,173.8708,-1.1760,-13176.5622
C01268=66.782,-49.709,76.575,173.6819,-0.0796,-13176.6621
C01269=60.870,-45.159,74.567,174.4737,-0.0632,-13176.5714
C01270=55.523,-41.042,71.901,175.7117,-0.1034,-13176.4714
C01271=51.344,-38.042,69.285,178.6998,-0.0933,-13176.5356
C01272=48.211,-36.955,67.386,-163.3536,14.5351,-13177.4711
C01273=45.408,-38.660,66.632,-173.6783,33.4962,-13180.4108
C01274=43.572,-40.607,66.599,179.7247,34.6655,-13182.9827
C01275=42.111,-42.111,66.621,180.0000,34.6557,-13185.0000
C01276=40.607,-43.571,66.599,-179.7195,34.6689,-13187.0166
C01277=38.659,-45.409,66.632,173.6775,33.4961,-13189.5906
C01278=36.955,-48.211,67.386,163.3501,14.5305,-13192.5289
C01279=38.042,-51.344,69.285,-178.6998,-0.0933,-13193.4644
C01280=41.042,-55.523,71.901,-175.7117,-0.1034,-13193.5286
C01281=45.159,-60.870,74.567,-174.4737,-0.0632,-13193.4286
C01282=49.709,-66.782,76.575,-173.6819,-0.0796,-13193.3379
C01283=53.692,-72.396,77.551,-173.8708,-1.1760,-13193.4378
C01284=54.731,-78.373,78.062,-177.0289,-2.6213,-13195.0719
C01285=52.567,-83.926,78.476,-179.2889,-1.7910,-13197.9391
C01286=47.632,-87.904,78.891,-179.9965,-0.1257,-13201.5483
C01287=41.489,-90.984,79.163,-179.9995,-0.0128,-13205.4869
C01288=34.998,-93.673,79.163,-179.9986,-0.0127,-13209.5134
C01289=28.477,-95.839,78.891,179.9987,-0.1251,-13213.4515
C01290=22.174,-96.515,78.476,179.2889,-1.7890,-13217.0610
C01291=16.717,-94.118,78.062,177.0287,-2.6199,-13219.9283
C01292=13.226,-89.158,77.551,173.8761,-1.1797,-13221.5621
C01293=12.073,-82.372,76.575,173.6811,-0.0780,-13221.6617
C01294=11.109,-74.974,74.567,174.4741,-0.0631,-13221.5717
C01295=10.239,-68.282,71.901,175.7112,-0.0994,-13221.4719
C01296=9.406,-63.206,69.285,178.7004,-0.0905,-13221.5356
C01297=7.959,-60.221,67.386,-163.3494,14.5335,-13222.4712
C01298=4.772,-59.445,66.632,-173.6798,33.4987,-13225.4104
C01299=2.097,-59.523,66.599,179.7230,34.6655,-13227.9823
C01300=0.000,-59.554,66.621,180.0000,34.6578,-13230.0000
C01301=-2.096,-59.523,66.599,-179.7223,34.6655,-13232.0167
C01302=-4.772,-59.445,66.632,173.6803,33.4939,-13234.5896
C01303=-7.959,-60.222,67.386,163.3494,14.5335,-13237.5286
C01304=-9.406,-63.206,69.285,-178.7004,-0.0905,-13238.4644
C01305=-10.239,-68.282,71.901,-175.7112,-0.0994,-13238.5281
C01306=-11.109,-74.974,74.567,-174.4741,-0.0631,-13238.4283
C01307=-12.073,-82.372,76.575,-173.6811,-0.0780,-13238.3383
C01308=-13.226,-89.158,77.551,-173.8761,-1.1797,-13238.4379
C01309=-16.717,-94.118,78.062,-177.0287,-2.6199,-13240.0717
C01310=-22.174,-96.515,78.476,-179.2889,-1.7890,-13242.9390
C01311=-28.477,-95.839,78.891,-179.9987,-0.1251,-13246.5485
C01312=-34.998,-93.673,79.163,179.9986,-0.0127,-13250.4866
C01313=-41.489,-90.984,79.163,179.9995,-0.0128,-13254.5131
C01314=-47.632,-87.904,78.891,179.9965,-0.1257,-13258.4517
C01315=-52.567,-83.926,78.476,179.2889,-1.7910,-13262.0609
C01316=-54.731,-78.373,78.062,177.0289,-2.6213,-13264.9281
C01317=-53.692,-72.396,77.551,173.8708,-1.1760,-13266.5622
C01318=-49.709,-66.782,76.575,173.6819,-0.0796,-13266.6621
C01319=-45.159,-60.870,74.567,174.4737,-0.0632,-13266.5714
C01320=-41.042,-55.523,71.901,175.7117,-0.1034,-13266.4714
C01321=-38.042,-51.344,69.285,178.6998,-0.0933,-13266.5356
C01322=-36.955,-48.211,67.386,-163.3536,14.5351,-13267.4711
C01323=-38.660,-45.408,66.632,-173.6783,33.4962,-13270.4108
C01324=-40.607,-43.572,66.599,179.7247,34.6655,-13272.9827
C01325=-42.111,-42.111,66.621,180.0000,34.6557,-13275.0000
C01326=-43.571,-40.607,66.599,-179.7195,34.6689,-13277.0166
C01327=-45.409,-38.659,66.632,173.6775,33.4961,-13279.5906
C01328=-48.211,-36.955,67.386,163.3501,14.5305,-13282.5289
C01329=-51.344,-38.042,69.285,-178.6998,-0.0933,-13283.4644
C01330=-55.523,-41.042,71.901,-175.7117,-0.1034,-13283.5286
C01331=-60.870,-45.159,74.567,-174.4737,-0.0632,-13283.4286
C01332=-66.782,-49.709,76.575,-173.6819,-0.0796,-13283.3379
C01333=-72.396,-53.692,77.551,-173.8708,-1.1760,-13283.4378
C01334=-78.373,-54.731,78.062,-177.0289,-2.6213,-13285.0719
C01335=-83.926,-52.567,78.476,-179.2889,-1.7910,-13287.9391
C01336=-87.904,-47.632,78.891,-179.9965,-0.1257,-13291.5483
C01337=-90.984,-41.489,79.163,-179.9995,-0.0128,-13295.4869
C01338=-93.673,-34.998,79.163,-179.9986,-0.0127,-13299.5134
C01339=-95.839,-28.477,78.891,179.9987,-0.1251,-13303.4515
C01340=-96.515,-22.174,78.476,179.2889,-1.7890,-13307.0610
C01341=-94.118,-16.717,78.062,177.0287,-2.6199,-13309.9283
C01342=-89.158,-13.226,77.551,173.8761,-1.1797,-13311.5621
C01343=-82.372,-12.073,76.575,173.6811,-0.0780,-13311.6617
C01344=-74.974,-11.109,74.567,174.4741,-0.0631,-13311.5717
C01345=-68.282,-10.239,71.901,175.7112,-0.0994,-13311.4719
C01346=-63.206,-9.406,69.285,178.7004,-0.0905,-13311.5356
C01347=-60.221,-7.959,67.386,-163.3494,14.5335,-13312.4712
C01348=-59.445,-4.772,66.632,-173.6798,33.4987,-13315.4104
C01349=-59.523,-2.097,66.599,179.7230,34.6655,-13317.9823
C01350=-59.554,0.000,66.621,-180.0000,34.6578,-13320.0000
C01351=-59.523,2.096,66.599,-179.7223,34.6655,-13322.0167
C01352=-59.445,4.772,66.632,173.6803,33.4939,-13324.5896
C01353=-60.222,7.959,67.386,163.3494,14.5335,-13327.5286
C01354=-63.206,9.406,69.285,-178.7004,-0.0905,-13328.4644
C01355=-68.282,10.239,71.901,-175.7112,-0.0994,-13328.5281
C01356=-74.974,11.109,74.567,-174.4741,-0.0631,-13328.4283
C01357=-82.372,12.073,76.575,-173.6811,-0.0780,-13328.3383
C01358=-89.158,13.226,77.551,-173.8761,-1.1797,-13328.4379
C01359=-94.118,16.717,78.062,-177.0287,-2.6199,-13330.0717
C01360=-96.515,22.174,78.476,-179.2889,-1.7890,-13332.9390
C01361=-95.839,28.477,78.891,-179.9987,-0.1251,-13336.5485
C01362=-93.673,34.998,79.163,179.9986,-0.0127,-13340.4866
C01363=-90.984,41.489,79.163,179.9995,-0.0128,-13344.5131
C01364=-87.904,47.632,78.891,179.9965,-0.1257,-13348.4517
C01365=-83.926,52.567,78.476,179.2889,-1.7910,-13352.0609
C01366=-78.373,54.731,78.062,177.0289,-2.6213,-13354.9281
C01367=-72.396,53.692,77.551,173.8708,-1.1760,-13356.5622
C01368=-66.782,49.709,76.575,173.6819,-0.0796,-13356.6621
C01369=-60.870,45.159,74.567,174.4737,-0.0632,-13356.5714
C01370=-55.523,41.042,71.901,175.7117,-0.1034,-13356.4714
C01371=-51.344,38.042,69.285,178.6998,-0.0933,-13356.5356
C01372=-48.211,36.955,67.386,-163.3536,14.5351,-13357.4711
C01373=-45.408,38.660,66.632,-173.6783,33.4962,-13360.4108
C01374=-43.572,40.607,66.599,179.7247,34.6655,-13362.9827
C01375=-42.111,42.111,66.621,-180.0000,34.6557,-13365.0000
C01376=-40.607,43.571,66.599,-179.7195,34.6689,-13367.0166
C01377=-38.659,45.409,66.632,173.6775,33.4961,-13369.5906
C01378=-36.955,48.211,67.386,163.3501,14.5305,-13372.5289
C01379=-38.042,51.344,69.285,-178.6998,-0.0933,-13373.4644
C01380=-41.042,55.523,71.901,-175.7117,-0.1034,-13373.5286
C01381=-45.159,60.870,74.567,-174.4737,-0.0632,-13373.4286
C01382=-49.709,66.782,76.575,-173.6819,-0.0796,-13373.3379
C01383=-53.692,72.396,77.551,-173.8708,-1.1760,-13373.4378
C01384=-54.731,78.373,78.062,-177.0289,-2.6213,-13375.0719
C01385=-52.567,83.926,78.476,-179.2889,-1.7910,-13377.9391
C01386=-47.632,87.904,78.891,-179.9965,-0.1257,-13381.5483
C01387=-41.489,90.984,79.163,-179.9995,-0.0128,-13385.4869
C01388=-34.998,93.673,79.163,-179.9986,-0.0127,-13389.5134
C01389=-28.477,95.839,78.891,179.9987,-0.1251,-13393.4515
C01390=-22.174,96.515,78.476,179.2889,-1.7890,-13397.0610
C01391=-16.717,94.118,78.062,177.0287,-2.6199,-13399.9283
C01392=-13.226,89.158,77.551,173.8761,-1.1797,-13401.5621
C01393=-12.073,82.372,76.575,173.6811,-0.0780,-13401.6617
C01394=-11.109,74.974,74.567,174.4741,-0.0631,-13401.5717
C01395=-10.239,68.282,71.901,175.7112,-0.0994,-13401.4719
C01396=-9.406,63.206,69.285,178.7004,-0.0905,-13401.5356
C01397=-7.959,60.222,67.386,-163.3494,14.5335,-13402.4714
C01398=-4.772,59.445,66.632,-173.6803,33.4939,-13405.4104
C01399=-2.096,59.523,66.599,179.7223,34.6655,-13407.9833
C01400=0.000,58.319,68.442,-180.0000,33.6424,-13410.0000
C01401=1.984,58.291,68.419,-179.7349,33.6528,-13411.9494
C01402=4.582,58.225,68.453,173.6435,32.4018,-13414.4996
C01403=7.730,59.058,69.238,164.1787,13.2130,-13417.4570
C01404=9.135,62.185,71.215,-178.3577,-0.1005,-13418.3570
C01405=9.949,67.473,73.927,-175.8025,-0.0826,-13418.3879
C01406=10.820,74.409,76.674,-174.7933,-0.0431,-13418.2735
C01407=11.787,82.032,78.729,-174.1646,-0.0547,-13418.1767
C01408=12.929,88.996,79.725,-174.3851,-1.0436,-13418.2659
C01409=16.445,94.085,80.245,-177.2659,-2.3820,-13419.9145
C01410=21.964,96.553,80.665,-179.3477,-1.6266,-13422.8156
C01411=28.347,95.882,81.086,179.9979,-0.1141,-13426.4700
C01412=34.955,93.690,81.363,179.9986,-0.0127,-13430.4601
C01413=41.532,90.965,81.363,179.9995,-0.0128,-13434.5401
C01414=47.755,87.843,81.086,179.9989,-0.1180,-13438.5303
C01415=52.743,83.804,80.665,179.3513,-1.6270,-13442.1847
C01416=54.900,78.157,80.245,177.2696,-2.3811,-13445.0854
C01417=53.787,72.072,79.725,174.3816,-1.0449,-13446.7338
C01418=49.670,66.340,78.729,174.1696,-0.0563,-13446.8229
C01419=44.964,60.266,76.674,174.7950,-0.0468,-13446.7263
C01420=40.676,54.746,73.927,175.8029,-0.0822,-13446.6122
C01421=37.512,50.430,71.215,178.3596,-0.0990,-13446.6435
C01422=36.294,47.226,69.238,-164.1774,13.2171,-13447.5429
C01423=37.931,44.411,68.453,-173.6447,32.4038,-13450.5003
C01424=39.816,42.621,68.419,179.7347,33.6545,-13453.0512
C01425=41.238,41.238,68.442,-180.0000,33.6466,-13455.0000
C01426=42.621,39.816,68.419,-179.7347,33.6545,-13456.9488
C01427=44.412,37.931,68.453,173.6400,32.4000,-13459.5003
C01428=47.226,36.294,69.238,164.1774,13.2171,-13462.4571
C01429=50.430,37.512,71.215,-178.3596,-0.0990,-13463.3565
C01430=54.746,40.676,73.927,-175.8029,-0.0822,-13463.3878
C01431=60.266,44.964,76.674,-174.7950,-0.0468,-13463.2737
C01432=66.340,49.670,78.729,-174.1696,-0.0563,-13463.1771
C01433=72.072,53.787,79.725,-174.3816,-1.0449,-13463.2662
C01434=78.157,54.900,80.245,-177.2696,-2.3811,-13464.9146
C01435=83.804,52.743,80.665,-179.3513,-1.6270,-13467.8153
C01436=87.843,47.755,81.086,-179.9989,-0.1180,-13471.4697
C01437=90.965,41.532,81.363,-179.9995,-0.0128,-13475.4599
C01438=93.690,34.955,81.363,-179.9986,-0.0127,-13479.5399
C01439=95.882,28.347,81.086,-179.9979,-0.1141,-13483.5300
C01440=96.553,21.964,80.665,179.3477,-1.6266,-13487.1844
C01441=94.085,16.445,80.245,177.2659,-2.3820,-13490.0855
C01442=88.996,12.929,79.725,174.3851,-1.0436,-13491.7341
C01443=82.032,11.787,78.729,174.1646,-0.0547,-13491.8233
C01444=74.409,10.820,76.674,174.7933,-0.0431,-13491.7265
C01445=67.473,9.949,73.927,175.8025,-0.0826,-13491.6121
C01446=62.185,9.135,71.215,178.3577,-0.1005,-13491.6430
C01447=59.058,7.730,69.238,-164.1787,13.2130,-13492.5430
C01448=58.225,4.582,68.453,-173.6435,32.4018,-13495.5004
C01449=58.291,1.984,68.419,179.7349,33.6528,-13498.0506
C01450=58.319,0.000,68.442,-180.0000,33.6424,-13500.0000
C01451=58.291,-1.983,68.419,-179.7342,33.6528,-13501.9484
C01452=58.225,-4.583,68.453,173.6429,32.4017,-13504.5006
C01453=59.058,-7.730,69.238,164.1787,13.2130,-13507.4570
C01454=62.185,-9.135,71.215,-178.3577,-0.1005,-13508.3570
C01455=67.473,-9.949,73.927,-175.8025,-0.0826,-13508.3879
C01456=74.409,-10.820,76.674,-174.7933,-0.0431,-13508.2735
C01457=82.032,-11.787,78.729,-174.1646,-0.0547,-13508.1767
C01458=88.996,-12.929,79.725,-174.3851,-1.0436,-13508.2659
C01459=94.085,-16.445,80.245,-177.2659,-2.3820,-13509.9145
C01460=96.553,-21.964,80.665,-179.3477,-1.6266,-13512.8156
C01461=95.882,-28.347,81.086,179.9979,-0.1141,-13516.4700
C01462=93.690,-34.955,81.363,179.9986,-0.0127,-13520.4601
C01463=90.965,-41.532,81.363,179.9995,-0.0128,-13524.5401
C01464=87.843,-47.755,81.086,179.9989,-0.1180,-13528.5303
C01465=83.804,-52.743,80.665,179.3513,-1.6270,-13532.1847
C01466=78.157,-54.900,80.245,177.2696,-2.3811,-13535.0854
C01467=72.072,-53.787,79.725,174.3816,-1.0449,-13536.7338
C01468=66.340,-49.670,78.729,174.1696,-0.0563,-13536.8229
C01469=60.266,-44.964,76.674,174.7950,-0.0468,-13536.7263
C01470=54.746,-40.676,73.927,175.8029,-0.0822,-13536.6122
C01471=50.430,-37.512,71.215,178.3596,-0.0990,-13536.6435
C01472=47.226,-36.294,69.238,-164.1774,13.2171,-13537.5429
C01473=44.411,-37.931,68.453,-173.6447,32.4038,-13540.5003
C01474=42.621,-39.816,68.419,179.7347,33.6545,-13543.0512
C01475=41.238,-41.238,68.442,-180.0000,33.6466,-13545.0000
C01476=39.816,-42.621,68.419,-179.7347,33.6545,-13546.9488
C01477=37.931,-44.412,68.453,173.6400,32.4000,-13549.5003
C01478=36.294,-47.226,69.238,164.1774,13.2171,-13552.4571
C01479=37.512,-50.430,71.215,-178.3596,-0.0990,-13553.3565
C01480=40.676,-54.746,73.927,-175.8029,-0.0822,-13553.3878
C01481=44.964,-60.266,76.674,-174.7950,-0.0468,-13553.2737
C01482=49.670,-66.340,78.729,-174.1696,-0.0563,-13553.1771
C01483=53.787,-72.072,79.725,-174.3816,-1.0449,-13553.2662
C01484=54.900,-78.157,80.245,-177.2696,-2.3811,-13554.9146
C01485=52.743,-83.804,80.665,-179.3513,-1.6270,-13557.8153
C01486=47.755,-87.843,81.086,-179.9989,-0.1180,-13561.4697
C01487=41.532,-90.965,81.363,-179.9995,-0.0128,-13565.4599
C01488=34.955,-93.690,81.363,-179.9986,-0.0127,-13569.5399
C01489=28.347,-95.882,81.086,-179.9979,-0.1141,-13573.5300
C01490=21.964,-96.553,80.665,179.3477,-1.6266,-13577.1844
C01491=16.445,-94.085,80.245,177.2659,-2.3820,-13580.0855
C01492=12.929,-88.996,79.725,174.3851,-1.0436,-13581.7341
C01493=11.787,-82.032,78.729,174.1646,-0.0547,-13581.8233
C01494=10.820,-74.409,76.674,174.7933,-0.0431,-13581.7265
C01495=9.949,-67.473,73.927,175.8025,-0.0826,-13581.6121
C01496=9.135,-62.185,71.215,178.3577,-0.1005,-13581.6430
C01497=7.730,-59.058,69.238,-164.1787,13.2130,-13582.5430
C01498=4.582,-58.225,68.453,-173.6435,32.4018,-13585.5004
C01499=1.984,-58.291,68.419,179.7349,33.6528,-13588.0506
C01500=0.000,-58.319,68.442,-180.0000,33.6424,-13590.0000
C01501=-1.983,-58.291,68.419,-179.7342,33.6528,-13591.9484
C01502=-4.583,-58.225,68.453,173.6429,32.4017,-13594.5006
C01503=-7.730,-59.058,69.238,164.1787,13.2130,-13597.4570
C01504=-9.135,-62.185,71.215,-178.3577,-0.1005,-13598.3570
C01505=-9.949,-67.473,73.927,-175.8025,-0.0826,-13598.3879
C01506=-10.820,-74.409,76.674,-174.7933,-0.0431,-13598.2735
C01507=-11.787,-82.032,78.729,-174.1646,-0.0547,-13598.1767
C01508=-12.929,-88.996,79.725,-174.3851,-1.0436,-13598.2659
C01509=-16.445,-94.085,80.245,-177.2659,-2.3820,-13599.9145
C01510=-21.964,-96.553,80.665,-179.3477,-1.6266,-13602.8156
C01511=-28.347,-95.882,81.086,179.9979,-0.1141,-13606.4700
C01512=-34.955,-93.690,81.363,179.9986,-0.0127,-13610.4601
C01513=-41.532,-90.965,81.363,179.9995,-0.0128,-13614.5401
C01514=-47.755,-87.843,81.086,179.9989,-0.1180,-13618.5303
C01515=-52.743,-83.804,80.665,179.3513,-1.6270,-13622.1847
C01516=-54.900,-78.157,80.245,177.2696,-2.3811,-13625.0854
C01517=-53.787,-72.072,79.725,174.3816,-1.0449,-13626.7338
C01518=-49.670,-66.340,78.729,174.1696,-0.0563,-13626.8229
C01519=-44.964,-60.266,76.674,174.7950,-0.0468,-13626.7263
C01520=-40.676,-54.746,73.927,175.8029,-0.0822,-13626.6122
C01521=-37.512,-50.430,71.215,178.3596,-0.0990,-13626.6435
C01522=-36.294,-47.226,69.238,-164.1774,13.2171,-13627.5429
C01523=-37.931,-44.411,68.453,-173.6447,32.4038,-13630.5003
C01524=-39.816,-42.621,68.419,179.7347,33.6545,-13633.0512
C01525=-41.238,-41.238,68.442,180.0000,33.6466,-13635.0000
C01526=-42.621,-39.816,68.419,-179.7347,33.6545,-13636.9488
C01527=-44.412,-37.931,68.453,173.6400,32.4000,-13639.5003
C01528=-47.226,-36.294,69.238,164.1774,13.2171,-13642.4571
C01529=-50.430,-37.512,71.215,-178.3596,-0.0990,-13643.3565
C01530=-54.746,-40.676,73.927,-175.8029,-0.0822,-13643.3878
C01531=-60.266,-44.964,76.674,-174.7950,-0.0468,-13643.2737
C01532=-66.340,-49.670,78.729,-174.1696,-0.0563,-13643.1771
C01533=-72.072,-53.787,79.725,-174.3816,-1.0449,-13643.2662
C01534=-78.157,-54.900,80.245,-177.2696,-2.3811,-13644.9146
C01535=-83.804,-52.743,80.665,-179.3513,-1.6270,-13647.8153
C01536=-87.843,-47.755,81.086,-179.9989,-0.1180,-13651.4697
C01537=-90.965,-41.532,81.363,-179.9995,-0.0128,-13655.4599
C01538=-93.690,-34.955,81.363,-179.9986,-0.0127,-13659.5399
C01539=-95.882,-28.347,81.086,-179.9979,-0.1141,-13663.5300
C01540=-96.553,-21.964,80.665,179.3477,-1.6266,-13667.1844
C01541=-94.085,-16.445,80.245,177.2659,-2.3820,-13670.0855
C01542=-88.996,-12.929,79.725,174.3851,-1.0436,-13671.7341
C01543=-82.032,-11.787,78.729,174.1646,-0.0547,-13671.8233
C01544=-74.409,-10.820,76.674,174.7933,-0.0431,-13671.7265
C01545=-67.473,-9.949,73.927,175.8025,-0.0826,-13671.6121
C01546=-62.185,-9.135,71.215,178.3577,-0.1005,-13671.6430
C01547=-59.058,-7.730,69.238,-164.1787,13.2130,-13672.5430
C01548=-58.225,-4.582,68.453,-173.6435,32.4018,-13675.5004
C01549=-58.291,-1.984,68.419,179.7349,33.6528,-13678.0506
C01550=-58.319,0.000,68.442,180.0000,33.6424,-13680.0000
C01551=-58.291,1.983,68.419,-179.7342,33.6528,-13681.9484
C01552=-58.225,4.583,68.453,173.6429,32.4017,-13684.5006
C01553=-59.058,7.730,69.238,164.1787,13.2130,-13687.4570
C01554=-62.185,9.135,71.215,-178.3577,-0.1005,-13688.3570
C01555=-67.473,9.949,73.927,-175.8025,-0.0826,-13688.3879
C01556=-74.409,10.820,76.674,-174.7933,-0.0431,-13688.2735
C01557=-82.032,11.787,78.729,-174.1646,-0.0547,-13688.1767
C01558=-88.996,12.929,79.725,-174.3851,-1.0436,-13688.2659
C01559=-94.085,16.445,80.245,-177.2659,-2.3820,-13689.9145
C01560=-96.553,21.964,80.665,-179.3477,-1.6266,-13692.8156
C01561=-95.882,28.347,81.086,179.9979,-0.1141,-13696.4700
C01562=-93.690,34.955,81.363,179.9986,-0.0127,-13700.4601
C01563=-90.965,41.532,81.363,179.9995,-0.0128,-13704.5401
C01564=-87.843,47.755,81.086,179.9989,-0.1180,-13708.5303
C01565=-83.804,52.743,80.665,179.3513,-1.6270,-13712.1847
C01566=-78.157,54.900,80.245,177.2696,-2.3811,-13715.0854
C01567=-72.072,53.787,79.725,174.3816,-1.0449,-13716.7338
C01568=-66.340,49.670,78.729,174.1696,-0.0563,-13716.8229
C01569=-60.266,44.964,76.674,174.7950,-0.0468,-13716.7263
C01570=-54.746,40.676,73.927,175.8029,-0.0822,-13716.6122
C01571=-50.430,37.512,71.215,178.3596,-0.0990,-13716.6435
C01572=-47.226,36.294,69.238,-164.1774,13.2171,-13717.5429
C01573=-44.411,37.931,68.453,-173.6447,32.4038,-13720.5003
C01574=-42.621,39.816,68.419,179.7347,33.6545,-13723.0512
C01575=-41.238,41.238,68.442,180.0000,33.6466,-13725.0000
C01576=-39.816,42.621,68.419,-179.7347,33.6545,-13726.9488
C01577=-37.931,44.412,68.453,173.6400,32.4000,-13729.5003
C01578=-36.294,47.226,69.238,164.1774,13.2171,-13732.4571
C01579=-37.512,50.430,71.215,-178.3596,-0.0990,-13733.3565
C01580=-40.676,54.746,73.927,-175.8029,-0.0822,-13733.3878
C01581=-44.964,60.266,76.674,-174.7950,-0.0468,-13733.2737
C01582=-49.670,66.340,78.729,-174.1696,-0.0563,-13733.1771
C01583=-53.787,72.072,79.725,-174.3816,-1.0449,-13733.2662
C01584=-54.900,78.157,80.245,-177.2696,-2.3811,-13734.9146
C01585=-52.743,83.804,80.665,-179.3513,-1.6270,-13737.8153
C01586=-47.755,87.843,81.086,-179.9989,-0.1180,-13741.4697
C01587=-41.532,90.965,81.363,-179.9995,-0.0128,-13745.4599
C01588=-34.955,93.690,81.363,-179.9986,-0.0127,-13749.5399
C01589=-28.347,95.882,81.086,-179.9979,-0.1141,-13753.5300
C01590=-21.964,96.553,80.665,179.3477,-1.6266,-13757.1844
C01591=-16.445,94.085,80.245,177.2659,-2.3820,-13760.0855
C01592=-12.929,88.996,79.725,174.3851,-1.0436,-13761.7341
C01593=-11.787,82.032,78.729,174.1646,-0.0547,-13761.8233
C01594=-10.820,74.409,76.674,174.7933,-0.0431,-13761.7265
C01595=-9.949,67.473,73.927,175.8025,-0.0826,-13761.6121
C01596=-9.135,62.185,71.215,178.3577,-0.1005,-13761.6430
C01597=-7.730,59.058,69.238,-164.1787,13.2130,-13762.5430
C01598=-4.583,58.225,68.453,-173.6429,32.4017,-13765.4994
C01599=-1.983,58.291,68.419,179.7342,33.6528,-13768.0516
C01600=0.000,57.118,70.285,-180.0000,32.4949,-13770.0000
C01601=1.874,57.094,70.261,-179.7573,32.5080,-13771.8799
C01602=4.398,57.039,70.297,173.6555,31.1772,-13774.4091
C01603=7.507,57.930,71.114,165.0758,11.9424,-13777.3837
C01604=8.875,61.204,73.167,-178.1043,-0.0957,-13778.2508
C01605=9.674,66.709,75.971,-175.9523,-0.0621,-13778.2514
C01606=10.553,73.885,78.794,-175.1749,-0.0294,-13778.1286
C01607=11.527,81.722,80.892,-174.7101,-0.0362,-13778.0287
C01608=12.662,88.851,81.904,-174.9556,-0.9120,-13778.1105
C01609=16.202,94.056,82.431,-177.5455,-2.1207,-13779.7738
C01610=21.776,96.587,82.857,-179.4149,-1.4483,-13782.7052
C01611=28.231,95.920,83.283,-180.0000,-0.1015,-13786.4001
C01612=34.916,93.705,83.562,179.9986,-0.0127,-13790.4362
C01613=41.570,90.949,83.562,179.9996,-0.0128,-13794.5637
C01614=47.863,87.788,83.283,179.9986,-0.1052,-13798.5997
C01615=52.900,83.695,82.857,179.4162,-1.4469,-13802.2952
C01616=55.051,77.964,82.431,177.5443,-2.1205,-13805.2262
C01617=53.873,71.781,81.904,174.9523,-0.9140,-13806.8889
C01618=49.635,65.937,80.892,174.7131,-0.0370,-13806.9711
C01619=44.783,59.707,78.794,175.1691,-0.0312,-13806.8716
C01620=40.330,54.011,75.971,175.9514,-0.0603,-13806.7487
C01621=37.003,49.553,73.167,178.1031,-0.0935,-13806.7500
C01622=35.654,46.271,71.114,-165.0753,11.9430,-13807.6160
C01623=37.223,43.442,70.297,-173.6602,31.1794,-13810.5914
C01624=39.047,41.697,70.261,179.7562,32.5069,-13813.1202
C01625=40.388,40.388,70.285,-180.0000,32.4978,-13815.0000
C01626=41.696,39.047,70.261,-179.7558,32.5069,-13816.8791
C01627=43.443,37.223,70.297,173.6555,31.1756,-13819.4092
C01628=46.271,35.654,71.114,165.0753,11.9430,-13822.3840
C01629=49.553,37.003,73.167,-178.1031,-0.0935,-13823.2500
C01630=54.011,40.330,75.971,-175.9514,-0.0603,-13823.2513
C01631=59.707,44.783,78.794,-175.1691,-0.0312,-13823.1284
C01632=65.937,49.635,80.892,-174.7131,-0.0370,-13823.0289
C01633=71.781,53.873,81.904,-174.9523,-0.9140,-13823.1111
C01634=77.964,55.051,82.431,-177.5443,-2.1205,-13824.7738
C01635=83.695,52.900,82.857,-179.4162,-1.4469,-13827.7048
C01636=87.788,47.863,83.283,-179.9986,-0.1052,-13831.4003
C01637=90.949,41.570,83.562,-179.9996,-0.0128,-13835.4363
C01638=93.705,34.916,83.562,-179.9986,-0.0127,-13839.5638
C01639=95.920,28.231,83.283,180.0000,-0.1015,-13843.5999
C01640=96.587,21.776,82.857,179.4149,-1.4483,-13847.2948
C01641=94.056,16.202,82.431,177.5455,-2.1207,-13850.2262
C01642=88.851,12.662,81.904,174.9556,-0.9120,-13851.8895
C01643=81.722,11.527,80.892,174.7101,-0.0362,-13851.9713
C01644=73.885,10.553,78.794,175.1749,-0.0294,-13851.8714
C01645=66.709,9.674,75.971,175.9523,-0.0621,-13851.7486
C01646=61.204,8.875,73.167,178.1043,-0.0957,-13851.7492
C01647=57.930,7.507,71.114,-165.0758,11.9424,-13852.6163
C01648=57.039,4.398,70.297,-173.6555,31.1772,-13855.5909
C01649=57.094,1.874,70.261,179.7573,32.5080,-13858.1201
C01650=57.118,0.000,70.285,-180.0000,32.4949,-13860.0000
C01651=57.094,-1.874,70.261,-179.7573,32.5080,-13861.8799
C01652=57.039,-4.398,70.297,173.6555,31.1772,-13864.4091
C01653=57.930,-7.507,71.114,165.0758,11.9424,-13867.3837
C01654=61.204,-8.875,73.167,-178.1043,-0.0957,-13868.2508
C01655=66.709,-9.674,75.971,-175.9523,-0.0621,-13868.2514
C01656=73.885,-10.553,78.794,-175.1749,-0.0294,-13868.1286
C01657=81.722,-11.527,80.892,-174.7101,-0.0362,-13868.0287
C01658=88.851,-12.662,81.904,-174.9556,-0.9120,-13868.1105
C01659=94.056,-16.202,82.431,-177.5455,-2.1207,-13869.7738
C01660=96.587,-21.776,82.857,-179.4149,-1.4483,-13872.7052
C01661=95.920,-28.231,83.283,-180.0000,-0.1015,-13876.4001
C01662=93.705,-34.916,83.562,179.9986,-0.0127,-13880.4362
C01663=90.949,-41.570,83.562,179.9996,-0.0128,-13884.5637
C01664=87.788,-47.863,83.283,179.9986,-0.1052,-13888.5997
C01665=83.695,-52.900,82.857,179.4162,-1.4469,-13892.2952
C01666=77.964,-55.051,82.431,177.5443,-2.1205,-13895.2262
C01667=71.781,-53.873,81.904,174.9523,-0.9140,-13896.8889
C01668=65.937,-49.635,80.892,174.7131,-0.0370,-13896.9711
C01669=59.707,-44.783,78.794,175.1691,-0.0312,-13896.8716
C01670=54.011,-40.330,75.971,175.9514,-0.0603,-13896.7487
C01671=49.553,-37.003,73.167,178.1031,-0.0935,-13896.7500
C01672=46.271,-35.654,71.114,-165.0753,11.9430,-13897.6160
C01673=43.442,-37.223,70.297,-173.6602,31.1794,-13900.5914
C01674=41.697,-39.047,70.261,179.7562,32.5069,-13903.1202
C01675=40.388,-40.388,70.285,-180.0000,32.4978,-13905.0000
C01676=39.047,-41.696,70.261,-179.7558,32.5069,-13906.8791
C01677=37.223,-43.443,70.297,173.6555,31.1756,-13909.4092
C01678=35.654,-46.271,71.114,165.0753,11.9430,-13912.3840
C01679=37.003,-49.553,73.167,-178.1031,-0.0935,-13913.2500
C01680=40.330,-54.011,75.971,-175.9514,-0.0603,-13913.2513
C01681=44.783,-59.707,78.794,-175.1691,-0.0312,-13913.1284
C01682=49.635,-65.937,80.892,-174.7131,-0.0370,-13913.0289
C01683=53.873,-71.781,81.904,-174.9523,-0.9140,-13913.1111
C01684=55.051,-77.964,82.431,-177.5443,-2.1205,-13914.7738
C01685=52.900,-83.695,82.857,-179.4162,-1.4469,-13917.7048
C01686=47.863,-87.788,83.283,-179.9986,-0.1052,-13921.4003
C01687=41.570,-90.949,83.562,-179.9996,-0.0128,-13925.4363
C01688=34.916,-93.705,83.562,-179.9986,-0.0127,-13929.5638
C01689=28.231,-95.920,83.283,180.0000,-0.1015,-13933.5999
C01690=21.776,-96.587,82.857,179.4149,-1.4483,-13937.2948
C01691=16.202,-94.056,82.431,177.5455,-2.1207,-13940.2262
C01692=12.662,-88.851,81.904,174.9556,-0.9120,-13941.8895
C01693=11.527,-81.722,80.892,174.7101,-0.0362,-13941.9713
C01694=10.553,-73.885,78.794,175.1749,-0.0294,-13941.8714
C01695=9.674,-66.709,75.971,175.9523,-0.0621,-13941.7486
C01696=8.875,-61.204,73.167,178.1043,-0.0957,-13941.7492
C01697=7.507,-57.930,71.114,-165.0758,11.9424,-13942.6163
C01698=4.398,-57.039,70.297,-173.6555,31.1772,-13945.5909
C01699=1.874,-57.094,70.261,179.7573,32.5080,-13948.1201
C01700=0.000,-57.118,70.285,-180.0000,32.4949,-13950.0000
C01701=-1.874,-57.094,70.261,-179.7573,32.5080,-13951.8799
C01702=-4.398,-57.039,70.297,173.6555,31.1772,-13954.4091
C01703=-7.507,-57.930,71.114,165.0758,11.9424,-13957.3837
C01704=-8.875,-61.204,73.167,-178.1043,-0.0957,-13958.2508
C01705=-9.674,-66.709,75.971,-175.9523,-0.0621,-13958.2514
C01706=-10.553,-73.885,78.794,-175.1749,-0.0294,-13958.1286
C01707=-11.527,-81.722,80.892,-174.7101,-0.0362,-13958.0287
C01708=-12.662,-88.851,81.904,-174.9556,-0.9120,-13958.1105
